LIN {X 0,Y 322.903,Z 1049.964,A -85,B 0,C 180,E1 13541.731,E2 13541.731} C_VEL
LIN {X 0,Y 332.533,Z 1032.411,A -85,B 0,C 180,E1 13538.987,E2 13538.987} C_VEL
LIN {X 0,Y 341.786,Z 1014.049,A -85,B 0,C 180,E1 13536.641,E2 13536.641} C_VEL
LIN {X 0,Y 350.913,Z 994.604,A -85,B 0,C 180,E1 13534.565,E2 13534.565} C_VEL
LIN {X 0,Y 358.946,Z 975.482,A -85,B 0,C 180,E1 13532.888,E2 13532.888} C_VEL
LIN {X 0,Y 366.893,Z 954.723,A -85,B 0,C 180,E1 13531.368,E2 13531.368} C_VEL
LIN {X 0,Y 373.86,Z 933.503,A -85,B 0,C 180,E1 13530.106,E2 13530.106} C_VEL
LIN {X 0,Y 380.358,Z 910.815,A -85,B 0,C 180,E1 13529.008,E2 13529.008} C_VEL
LIN {X 0,Y 385.815,Z 887.235,A -85,B 0,C 180,E1 13528.129,E2 13528.129} C_VEL
LIN {X 0,Y 390.273,Z 863.229,A -85,B 0,C 180,E1 13527.442,E2 13527.442} C_VEL
LIN {X 0,Y 393.285,Z 839.012,A -85,B 0,C 180,E1 13526.936,E2 13526.936} C_VEL
LIN {X 0,Y 410.602,Z 627.439,A -85,B 0,C 180,E1 13523.387,E2 13523.387} C_VEL
LIN {X 0,Y 404.165,Z 615.635,A -85,B 0,C 180,E1 13520.832,E2 13520.832} C_VEL
LIN {X 0,Y 397.85,Z 604.757,A -85,B 0,C 180,E1 13517.969,E2 13517.969} C_VEL
LIN {X 0,Y 392.489,Z 596.179,A -85,B 0,C 180,E1 13515.137,E2 13515.137} C_VEL
LIN {X 0,Y 387.858,Z 589.138,A -85,B 0,C 180,E1 13512.204,E2 13512.204} C_VEL
LIN {X 0,Y 384.835,Z 584.731,A -85,B 0,C 180,E1 13509.874,E2 13509.874} C_VEL
LIN {X 0,Y 381.69,Z 580.189,A -85,B 0,C 180,E1 13506.77,E2 13506.77} C_VEL
LIN {X 0,Y 378.64,Z 576.347,A -85,B 0,C 180,E1 13501.816,E2 13501.816} C_VEL
LIN {X 0,Y 377.972,Z 575.706,A -85,B 0,C 180,E1 13498.787,E2 13498.787} C_VEL
LIN {X 0,Y 378.254,Z 577.065,A -85,B 0,C 180,E1 13495.3,E2 13495.3} C_VEL
LIN {X 0,Y 380.09,Z 579.956,A -85,B 0,C 180,E1 13491.376,E2 13491.376} C_VEL
LIN {X 0,Y 382.905,Z 585.008,A -85,B 0,C 180,E1 13487.942,E2 13487.942} C_VEL
LIN {X 0,Y 385.173,Z 588.932,A -85,B 0,C 180,E1 13485.876,E2 13485.876} C_VEL
LIN {X 0,Y 388.941,Z 595.206,A -85,B 0,C 180,E1 13483.112,E2 13483.112} C_VEL
LIN {X 0,Y 394.171,Z 604.5,A -85,B 0,C 180,E1 13479.973,E2 13479.973} C_VEL
LIN {X 0,Y 400.396,Z 616.098,A -85,B 0,C 180,E1 13476.878,E2 13476.878} C_VEL
LIN {X 0,Y 406.234,Z 627.647,A -85,B 0,C 180,E1 13474.368,E2 13474.368} C_VEL
LIN {X 0,Y 409.258,Z 634.08,A -85,B 0,C 180,E1 13473.169,E2 13473.169} C_VEL
LIN {X 0,Y 392.663,Z 845.729,A -85,B 0,C 180,E1 13469.732,E2 13469.732} C_VEL
LIN {X 0,Y 389.223,Z 870.537,A -85,B 0,C 180,E1 13469.186,E2 13469.186} C_VEL
LIN {X 0,Y 384.954,Z 892.745,A -85,B 0,C 180,E1 13468.528,E2 13468.528} C_VEL
LIN {X 0,Y 379.397,Z 915.306,A -85,B 0,C 180,E1 13467.637,E2 13467.637} C_VEL
LIN {X 0,Y 373.122,Z 936.697,A -85,B 0,C 180,E1 13466.575,E2 13466.575} C_VEL
LIN {X 0,Y 365.655,Z 958.094,A -85,B 0,C 180,E1 13465.237,E2 13465.237} C_VEL
LIN {X 0,Y 357.495,Z 978.757,A -85,B 0,C 180,E1 13463.661,E2 13463.661} C_VEL
LIN {X 0,Y 348.897,Z 997.813,A -85,B 0,C 180,E1 13461.863,E2 13461.863} C_VEL
LIN {X 0,Y 339.99,Z 1016.009,A -85,B 0,C 180,E1 13459.8,E2 13459.8} C_VEL
LIN {X 0,Y 330.683,Z 1033.179,A -85,B 0,C 180,E1 13457.415,E2 13457.415} C_VEL
LIN {X 0,Y 321.318,Z 1049.45,A -85,B 0,C 180,E1 13454.691,E2 13454.691} C_VEL
LIN {X 0,Y 312.434,Z 1063.871,A -85,B 0,C 180,E1 13451.734,E2 13451.734} C_VEL
LIN {X 0,Y 303.544,Z 1077.822,A -85,B 0,C 180,E1 13448.264,E2 13448.264} C_VEL
LIN {X 0,Y 296.111,Z 1089.153,A -85,B 0,C 180,E1 13444.797,E2 13444.797} C_VEL
LIN {X 0,Y 288.785,Z 1100.377,A -85,B 0,C 180,E1 13440.596,E2 13440.596} C_VEL
LIN {X 0,Y 283.114,Z 1109.26,A -85,B 0,C 180,E1 13436.424,E2 13436.424} C_VEL
LIN {X 0,Y 278.099,Z 1117.701,A -85,B 0,C 180,E1 13431.373,E2 13431.373} C_VEL
LIN {X 0,Y 275.121,Z 1123.417,A -85,B 0,C 180,E1 13426.903,E2 13426.903} C_VEL
LIN {X 0,Y 273.116,Z 1128.104,A -85,B 0,C 180,E1 13421.831,E2 13421.831} C_VEL
LIN {X 0,Y 272.314,Z 1130.762,A -85,B 0,C 180,E1 13417.52,E2 13417.52} C_VEL
LIN {X 0,Y 272.028,Z 1132.355,A -85,B 0,C 180,E1 13412.739,E2 13412.739} C_VEL
LIN {X 0,Y 272.01,Z 1132.518,A -85,B 0,C 180,E1 13408.736,E2 13408.736} C_VEL
LIN {X 0,Y 272.117,Z 1131.71,A -85,B 0,C 180,E1 13404.729,E2 13404.729} C_VEL
LIN {X 0,Y 272.676,Z 1129.578,A -85,B 0,C 180,E1 13400.076,E2 13400.076} C_VEL
LIN {X 0,Y 274.088,Z 1125.684,A -85,B 0,C 180,E1 13395.205,E2 13395.205} C_VEL
LIN {X 0,Y 276.732,Z 1120.334,A -85,B 0,C 180,E1 13390.365,E2 13390.365} C_VEL
LIN {X 0,Y 280.577,Z 1113.483,A -85,B 0,C 180,E1 13385.806,E2 13385.806} C_VEL
LIN {X 0,Y 285.829,Z 1105.112,A -85,B 0,C 180,E1 13381.363,E2 13381.363} C_VEL
LIN {X 0,Y 292.154,Z 1095.285,A -85,B 0,C 180,E1 13377.265,E2 13377.265} C_VEL
LIN {X 0,Y 299.769,Z 1083.78,A -85,B 0,C 180,E1 13373.34,E2 13373.34} C_VEL
LIN {X 0,Y 307.712,Z 1071.486,A -85,B 0,C 180,E1 13369.955,E2 13369.955} C_VEL
LIN {X 0,Y 316.612,Z 1057.407,A -85,B 0,C 180,E1 13366.74,E2 13366.74} C_VEL
LIN {X 0,Y 325.483,Z 1042.519,A -85,B 0,C 180,E1 13363.97,E2 13363.97} C_VEL
LIN {X 0,Y 334.935,Z 1025.814,A -85,B 0,C 180,E1 13361.385,E2 13361.385} C_VEL
LIN {X 0,Y 343.865,Z 1008.56,A -85,B 0,C 180,E1 13359.201,E2 13359.201} C_VEL
LIN {X 0,Y 353.149,Z 989.023,A -85,B 0,C 180,E1 13357.153,E2 13357.153} C_VEL
LIN {X 0,Y 361.054,Z 970.43,A -85,B 0,C 180,E1 13355.561,E2 13355.561} C_VEL
LIN {X 0,Y 369.229,Z 948.778,A -85,B 0,C 180,E1 13354.038,E2 13354.038} C_VEL
LIN {X 0,Y 375.381,Z 929.911,A -85,B 0,C 180,E1 13352.959,E2 13352.959} C_VEL
LIN {X 0,Y 381.682,Z 907.48,A -85,B 0,C 180,E1 13351.92,E2 13351.92} C_VEL
LIN {X 0,Y 386.562,Z 885.839,A -85,B 0,C 180,E1 13351.142,E2 13351.142} C_VEL
LIN {X 0,Y 390.855,Z 861.566,A -85,B 0,C 180,E1 13350.489,E2 13350.489} C_VEL
LIN {X 0,Y 393.474,Z 839.331,A -85,B 0,C 180,E1 13350.048,E2 13350.048} C_VEL
LIN {X 0,Y 401.911,Z 730.436,A -85,B 0,C 180,E1 13348.274,E2 13348.274} C_VEL
LIN {X 0,Y 402.052,Z 722.869,A -85,B 0,C 180,E1 13348.025,E2 13348.025} C_VEL
LIN {X 0,Y 400.861,Z 703.163,A -85,B 0,C 180,E1 13346.9,E2 13346.9} C_VEL
LIN {X 0,Y 401.076,Z 696.654,A -85,B 0,C 180,E1 13346.702,E2 13346.702} C_VEL
LIN {X 0,Y 405.736,Z 638.185,A -85,B 0,C 180,E1 13345.744,E2 13345.744} C_VEL
LIN {X 0,Y 400.125,Z 626.654,A -85,B 0,C 180,E1 13343.334,E2 13343.334} C_VEL
LIN {X 0,Y 395.257,Z 617.143,A -85,B 0,C 180,E1 13340.975,E2 13340.975} C_VEL
LIN {X 0,Y 391.098,Z 609.419,A -85,B 0,C 180,E1 13338.676,E2 13338.676} C_VEL
LIN {X 0,Y 386.949,Z 601.81,A -85,B 0,C 180,E1 13335.974,E2 13335.974} C_VEL
LIN {X 0,Y 382.739,Z 594.401,A -85,B 0,C 180,E1 13332.523,E2 13332.523} C_VEL
LIN {X 0,Y 380.657,Z 590.854,A -85,B 0,C 180,E1 13330.289,E2 13330.289} C_VEL
LIN {X 0,Y 378.767,Z 587.132,A -85,B 0,C 180,E1 13327.432,E2 13327.432} C_VEL
LIN {X 0,Y 377.279,Z 584.215,A -85,B 0,C 180,E1 13321.974,E2 13321.974} C_VEL
LIN {X 0,Y 377.726,Z 584.352,A -85,B 0,C 180,E1 13318.938,E2 13318.938} C_VEL
LIN {X 0,Y 379.196,Z 586.5,A -85,B 0,C 180,E1 13315.614,E2 13315.614} C_VEL
LIN {X 0,Y 381.242,Z 588.925,A -85,B 0,C 180,E1 13312.919,E2 13312.919} C_VEL
LIN {X 0,Y 384.711,Z 594.101,A -85,B 0,C 180,E1 13309.593,E2 13309.593} C_VEL
LIN {X 0,Y 387.934,Z 599.004,A -85,B 0,C 180,E1 13307.193,E2 13307.193} C_VEL
LIN {X 0,Y 392.201,Z 605.658,A -85,B 0,C 180,E1 13304.549,E2 13304.549} C_VEL
LIN {X 0,Y 397.939,Z 615.402,A -85,B 0,C 180,E1 13301.543,E2 13301.543} C_VEL
LIN {X 0,Y 403.54,Z 625.439,A -85,B 0,C 180,E1 13299.02,E2 13299.02} C_VEL
LIN {X 0,Y 407.083,Z 632.137,A -85,B 0,C 180,E1 13297.567,E2 13297.567} C_VEL
LIN {X 0,Y 389.262,Z 843.506,A -85,B 0,C 180,E1 13294.032,E2 13294.032} C_VEL
LIN {X 0,Y 385.581,Z 869.279,A -85,B 0,C 180,E1 13293.455,E2 13293.455} C_VEL
LIN {X 0,Y 381.197,Z 891.496,A -85,B 0,C 180,E1 13292.795,E2 13292.795} C_VEL
LIN {X 0,Y 375.18,Z 915.552,A -85,B 0,C 180,E1 13291.854,E2 13291.854} C_VEL
LIN {X 0,Y 368.839,Z 936.823,A -85,B 0,C 180,E1 13290.8,E2 13290.8} C_VEL
LIN {X 0,Y 360.787,Z 959.799,A -85,B 0,C 180,E1 13289.376,E2 13289.376} C_VEL
LIN {X 0,Y 352.95,Z 979.483,A -85,B 0,C 180,E1 13287.893,E2 13287.893} C_VEL
LIN {X 0,Y 343.751,Z 1000.055,A -85,B 0,C 180,E1 13285.996,E2 13285.996} C_VEL
LIN {X 0,Y 334.941,Z 1018.035,A -85,B 0,C 180,E1 13284,E2 13284} C_VEL
LIN {X 0,Y 324.794,Z 1037.02,A -85,B 0,C 180,E1 13281.44,E2 13281.44} C_VEL
LIN {X 0,Y 315.852,Z 1052.706,A -85,B 0,C 180,E1 13278.889,E2 13278.889} C_VEL
LIN {X 0,Y 305.817,Z 1069.374,A -85,B 0,C 180,E1 13275.598,E2 13275.598} C_VEL
LIN {X 0,Y 297.663,Z 1082.472,A -85,B 0,C 180,E1 13272.469,E2 13272.469} C_VEL
LIN {X 0,Y 288.631,Z 1096.717,A -85,B 0,C 180,E1 13268.324,E2 13268.324} C_VEL
LIN {X 0,Y 281.666,Z 1107.82,A -85,B 0,C 180,E1 13264.363,E2 13264.363} C_VEL
LIN {X 0,Y 275.153,Z 1118.6,A -85,B 0,C 180,E1 13259.618,E2 13259.618} C_VEL
LIN {X 0,Y 270.803,Z 1126.415,A -85,B 0,C 180,E1 13255.36,E2 13255.36} C_VEL
LIN {X 0,Y 267.019,Z 1134.293,A -85,B 0,C 180,E1 13249.923,E2 13249.923} C_VEL
LIN {X 0,Y 265.197,Z 1139.135,A -85,B 0,C 180,E1 13245.527,E2 13245.527} C_VEL
LIN {X 0,Y 264.211,Z 1143.133,A -85,B 0,C 180,E1 13240.687,E2 13240.687} C_VEL
LIN {X 0,Y 263.966,Z 1145.544,A -85,B 0,C 180,E1 13235.87,E2 13235.87} C_VEL
LIN {X 0,Y 263.989,Z 1146.491,A -85,B 0,C 180,E1 13231.954,E2 13231.954} C_VEL
LIN {X 0,Y 263.992,Z 1146.511,A -85,B 0,C 180,E1 13228.264,E2 13228.264} C_VEL
LIN {X 0,Y 263.96,Z 1145.604,A -85,B 0,C 180,E1 13224.348,E2 13224.348} C_VEL
LIN {X 0,Y 264.164,Z 1143.39,A -85,B 0,C 180,E1 13219.752,E2 13219.752} C_VEL
LIN {X 0,Y 265.132,Z 1139.314,A -85,B 0,C 180,E1 13214.693,E2 13214.693} C_VEL
LIN {X 0,Y 267.017,Z 1134.249,A -85,B 0,C 180,E1 13210.076,E2 13210.076} C_VEL
LIN {X 0,Y 270.611,Z 1126.713,A -85,B 0,C 180,E1 13204.854,E2 13204.854} C_VEL
LIN {X 0,Y 275.146,Z 1118.526,A -85,B 0,C 180,E1 13200.381,E2 13200.381} C_VEL
LIN {X 0,Y 281.976,Z 1107.201,A -85,B 0,C 180,E1 13195.433,E2 13195.433} C_VEL
LIN {X 0,Y 289.002,Z 1096.026,A -85,B 0,C 180,E1 13191.481,E2 13191.481} C_VEL
LIN {X 0,Y 297.648,Z 1082.336,A -85,B 0,C 180,E1 13187.528,E2 13187.528} C_VEL
LIN {X 0,Y 306.039,Z 1068.835,A -85,B 0,C 180,E1 13184.314,E2 13184.314} C_VEL
LIN {X 0,Y 316.373,Z 1051.575,A -85,B 0,C 180,E1 13180.943,E2 13180.943} C_VEL
LIN {X 0,Y 325.579,Z 1035.387,A -85,B 0,C 180,E1 13178.343,E2 13178.343} C_VEL
LIN {X 0,Y 335.535,Z 1016.541,A -85,B 0,C 180,E1 13175.849,E2 13175.849} C_VEL
LIN {X 0,Y 344.173,Z 998.833,A -85,B 0,C 180,E1 13173.904,E2 13173.904} C_VEL
LIN {X 0,Y 353.597,Z 977.481,A -85,B 0,C 180,E1 13171.969,E2 13171.969} C_VEL
LIN {X 0,Y 361.109,Z 958.494,A -85,B 0,C 180,E1 13170.554,E2 13170.554} C_VEL
LIN {X 0,Y 369.167,Z 935.183,A -85,B 0,C 180,E1 13169.132,E2 13169.132} C_VEL
LIN {X 0,Y 375.263,Z 914.581,A -85,B 0,C 180,E1 13168.121,E2 13168.121} C_VEL
LIN {X 0,Y 381.465,Z 889.296,A -85,B 0,C 180,E1 13167.15,E2 13167.15} C_VEL
LIN {X 0,Y 385.776,Z 867.055,A -85,B 0,C 180,E1 13166.502,E2 13166.502} C_VEL
LIN {X 0,Y 389.241,Z 841.731,A -85,B 0,C 180,E1 13165.95,E2 13165.95} C_VEL
LIN {X 0,Y 406.871,Z 631.81,A -85,B 0,C 180,E1 13162.432,E2 13162.432} C_VEL
LIN {X 0,Y 399.929,Z 619.065,A -85,B 0,C 180,E1 13159.498,E2 13159.498} C_VEL
LIN {X 0,Y 393.816,Z 608.454,A -85,B 0,C 180,E1 13156.483,E2 13156.483} C_VEL
LIN {X 0,Y 388.661,Z 600.303,A -85,B 0,C 180,E1 13153.464,E2 13153.464} C_VEL
LIN {X 0,Y 386.042,Z 596.274,A -85,B 0,C 180,E1 13151.656,E2 13151.656} C_VEL
LIN {X 0,Y 383.497,Z 592.425,A -85,B 0,C 180,E1 13149.606,E2 13149.606} C_VEL
LIN {X 0,Y 380.576,Z 588.062,A -85,B 0,C 180,E1 13146.638,E2 13146.638} C_VEL
LIN {X 0,Y 377.61,Z 584.234,A -85,B 0,C 180,E1 13141.669,E2 13141.669} C_VEL
LIN {X 0,Y 376.986,Z 583.655,A -85,B 0,C 180,E1 13138.632,E2 13138.632} C_VEL
LIN {X 0,Y 377.318,Z 585.14,A -85,B 0,C 180,E1 13135.135,E2 13135.135} C_VEL
LIN {X 0,Y 378.967,Z 587.768,A -85,B 0,C 180,E1 13131.58,E2 13131.58} C_VEL
LIN {X 0,Y 381.708,Z 592.841,A -85,B 0,C 180,E1 13128.133,E2 13128.133} C_VEL
LIN {X 0,Y 383.842,Z 596.653,A -85,B 0,C 180,E1 13126.134,E2 13126.134} C_VEL
LIN {X 0,Y 387.417,Z 602.767,A -85,B 0,C 180,E1 13123.43,E2 13123.43} C_VEL
LIN {X 0,Y 392.719,Z 612.462,A -85,B 0,C 180,E1 13120.168,E2 13120.168} C_VEL
LIN {X 0,Y 398.552,Z 623.768,A -85,B 0,C 180,E1 13117.194,E2 13117.194} C_VEL
LIN {X 0,Y 403.876,Z 634.566,A -85,B 0,C 180,E1 13114.836,E2 13114.836} C_VEL
LIN {X 0,Y 405.574,Z 638.42,A -85,B 0,C 180,E1 13114.126,E2 13114.126} C_VEL
LIN {X 0,Y 388.882,Z 845.735,A -85,B 0,C 180,E1 13110.768,E2 13110.768} C_VEL
LIN {X 0,Y 385.368,Z 870.544,A -85,B 0,C 180,E1 13110.226,E2 13110.226} C_VEL
LIN {X 0,Y 381.009,Z 892.763,A -85,B 0,C 180,E1 13109.574,E2 13109.574} C_VEL
LIN {X 0,Y 375.184,Z 915.866,A -85,B 0,C 180,E1 13108.667,E2 13108.667} C_VEL
LIN {X 0,Y 368.789,Z 937.151,A -85,B 0,C 180,E1 13107.614,E2 13107.614} C_VEL
LIN {X 0,Y 361.097,Z 958.617,A -85,B 0,C 180,E1 13106.274,E2 13106.274} C_VEL
LIN {X 0,Y 352.79,Z 979.102,A -85,B 0,C 180,E1 13104.713,E2 13104.713} C_VEL
LIN {X 0,Y 344.01,Z 998.066,A -85,B 0,C 180,E1 13102.926,E2 13102.926} C_VEL
LIN {X 0,Y 334.655,Z 1016.609,A -85,B 0,C 180,E1 13100.816,E2 13100.816} C_VEL
LIN {X 0,Y 325.255,Z 1033.454,A -85,B 0,C 180,E1 13098.466,E2 13098.466} C_VEL
LIN {X 0,Y 315.594,Z 1049.705,A -85,B 0,C 180,E1 13095.728,E2 13095.728} C_VEL
LIN {X 0,Y 306.483,Z 1064.007,A -85,B 0,C 180,E1 13092.772,E2 13092.772} C_VEL
LIN {X 0,Y 297.185,Z 1078.057,A -85,B 0,C 180,E1 13089.237,E2 13089.237} C_VEL
LIN {X 0,Y 289.444,Z 1089.384,A -85,B 0,C 180,E1 13085.719,E2 13085.719} C_VEL
LIN {X 0,Y 281.786,Z 1100.601,A -85,B 0,C 180,E1 13081.441,E2 13081.441} C_VEL
LIN {X 0,Y 275.83,Z 1109.483,A -85,B 0,C 180,E1 13077.178,E2 13077.178} C_VEL
LIN {X 0,Y 270.645,Z 1117.731,A -85,B 0,C 180,E1 13072.138,E2 13072.138} C_VEL
LIN {X 0,Y 267.456,Z 1123.446,A -85,B 0,C 180,E1 13067.574,E2 13067.574} C_VEL
LIN {X 0,Y 265.208,Z 1128.316,A -85,B 0,C 180,E1 13062.189,E2 13062.189} C_VEL
LIN {X 0,Y 264.353,Z 1130.934,A -85,B 0,C 180,E1 13057.826,E2 13057.826} C_VEL
LIN {X 0,Y 264.038,Z 1132.544,A -85,B 0,C 180,E1 13053.039,E2 13053.039} C_VEL
LIN {X 0,Y 264.013,Z 1132.728,A -85,B 0,C 180,E1 13048.698,E2 13048.698} C_VEL
LIN {X 0,Y 264.13,Z 1131.92,A -85,B 0,C 180,E1 13044.569,E2 13044.569} C_VEL
LIN {X 0,Y 264.728,Z 1129.79,A -85,B 0,C 180,E1 13039.775,E2 13039.775} C_VEL
LIN {X 0,Y 266.256,Z 1125.898,A -85,B 0,C 180,E1 13034.759,E2 13034.759} C_VEL
LIN {X 0,Y 269.081,Z 1120.55,A -85,B 0,C 180,E1 13029.783,E2 13029.783} C_VEL
LIN {X 0,Y 273.156,Z 1113.7,A -85,B 0,C 180,E1 13025.105,E2 13025.105} C_VEL
LIN {X 0,Y 278.688,Z 1105.334,A -85,B 0,C 180,E1 13020.558,E2 13020.558} C_VEL
LIN {X 0,Y 285.316,Z 1095.51,A -85,B 0,C 180,E1 13016.378,E2 13016.378} C_VEL
LIN {X 0,Y 293.265,Z 1084.013,A -85,B 0,C 180,E1 13012.388,E2 13012.388} C_VEL
LIN {X 0,Y 301.516,Z 1071.722,A -85,B 0,C 180,E1 13008.958,E2 13008.958} C_VEL
LIN {X 0,Y 310.74,Z 1057.658,A -85,B 0,C 180,E1 13005.712,E2 13005.712} C_VEL
LIN {X 0,Y 319.752,Z 1043.028,A -85,B 0,C 180,E1 13002.967,E2 13002.967} C_VEL
LIN {X 0,Y 329.453,Z 1026.447,A -85,B 0,C 180,E1 13000.378,E2 13000.378} C_VEL
LIN {X 0,Y 338.819,Z 1008.855,A -85,B 0,C 180,E1 12998.143,E2 12998.143} C_VEL
LIN {X 0,Y 348.023,Z 990.085,A -85,B 0,C 180,E1 12996.164,E2 12996.164} C_VEL
LIN {X 0,Y 356.36,Z 970.988,A -85,B 0,C 180,E1 12994.526,E2 12994.526} C_VEL
LIN {X 0,Y 364.462,Z 950.207,A -85,B 0,C 180,E1 12993.056,E2 12993.056} C_VEL
LIN {X 0,Y 371.092,Z 930.392,A -85,B 0,C 180,E1 12991.923,E2 12991.923} C_VEL
LIN {X 0,Y 377.525,Z 908.106,A -85,B 0,C 180,E1 12990.893,E2 12990.893} C_VEL
LIN {X 0,Y 382.609,Z 886.081,A -85,B 0,C 180,E1 12990.105,E2 12990.105} C_VEL
LIN {X 0,Y 386.974,Z 862.046,A -85,B 0,C 180,E1 12989.461,E2 12989.461} C_VEL
LIN {X 0,Y 389.69,Z 839.602,A -85,B 0,C 180,E1 12989.017,E2 12989.017} C_VEL
LIN {X 0,Y 401.076,Z 696.654,A -85,B 0,C 180,E1 12986.702,E2 12986.702} C_VEL
LIN {X 0,Y 401.28,Z 689.088,A -85,B 0,C 180,E1 12986.456,E2 12986.456} C_VEL
LIN {X 0,Y 400.308,Z 669.401,A -85,B 0,C 180,E1 12985.318,E2 12985.318} C_VEL
LIN {X 0,Y 400.547,Z 662.896,A -85,B 0,C 180,E1 12985.115,E2 12985.115} C_VEL
LIN {X 0,Y 402.173,Z 642.482,A -85,B 0,C 180,E1 12984.767,E2 12984.767} C_VEL
LIN {X 0,Y 396.956,Z 631.632,A -85,B 0,C 180,E1 12982.395,E2 12982.395} C_VEL
LIN {X 0,Y 392.14,Z 622.064,A -85,B 0,C 180,E1 12979.902,E2 12979.902} C_VEL
LIN {X 0,Y 387.97,Z 614.013,A -85,B 0,C 180,E1 12977.395,E2 12977.395} C_VEL
LIN {X 0,Y 384.024,Z 606.829,A -85,B 0,C 180,E1 12974.552,E2 12974.552} C_VEL
LIN {X 0,Y 381.229,Z 601.727,A -85,B 0,C 180,E1 12972.035,E2 12972.035} C_VEL
LIN {X 0,Y 379.441,Z 598.565,A -85,B 0,C 180,E1 12970.016,E2 12970.016} C_VEL
LIN {X 0,Y 377.634,Z 594.913,A -85,B 0,C 180,E1 12967.149,E2 12967.149} C_VEL
LIN {X 0,Y 376.306,Z 592.121,A -85,B 0,C 180,E1 12961.827,E2 12961.827} C_VEL
LIN {X 0,Y 376.75,Z 592.304,A -85,B 0,C 180,E1 12958.936,E2 12958.936} C_VEL
LIN {X 0,Y 378.309,Z 594.631,A -85,B 0,C 180,E1 12955.452,E2 12955.452} C_VEL
LIN {X 0,Y 380.058,Z 596.726,A -85,B 0,C 180,E1 12953.125,E2 12953.125} C_VEL
LIN {X 0,Y 383.355,Z 601.786,A -85,B 0,C 180,E1 12949.86,E2 12949.86} C_VEL
LIN {X 0,Y 386.504,Z 606.712,A -85,B 0,C 180,E1 12947.449,E2 12947.449} C_VEL
LIN {X 0,Y 390.619,Z 613.327,A -85,B 0,C 180,E1 12944.827,E2 12944.827} C_VEL
LIN {X 0,Y 396.255,Z 623.12,A -85,B 0,C 180,E1 12941.804,E2 12941.804} C_VEL
LIN {X 0,Y 402.628,Z 634.926,A -85,B 0,C 180,E1 12938.894,E2 12938.894} C_VEL
LIN {X 0,Y 403.466,Z 636.791,A -85,B 0,C 180,E1 12938.529,E2 12938.529} C_VEL
LIN {X 0,Y 385.611,Z 843.606,A -85,B 0,C 180,E1 12935.087,E2 12935.087} C_VEL
LIN {X 0,Y 381.867,Z 869.298,A -85,B 0,C 180,E1 12934.516,E2 12934.516} C_VEL
LIN {X 0,Y 377.399,Z 891.516,A -85,B 0,C 180,E1 12933.863,E2 12933.863} C_VEL
LIN {X 0,Y 371.534,Z 914.61,A -85,B 0,C 180,E1 12932.975,E2 12932.975} C_VEL
LIN {X 0,Y 365.305,Z 935.197,A -85,B 0,C 180,E1 12931.974,E2 12931.974} C_VEL
LIN {X 0,Y 357.061,Z 958.492,A -85,B 0,C 180,E1 12930.564,E2 12930.564} C_VEL
LIN {X 0,Y 349.366,Z 977.477,A -85,B 0,C 180,E1 12929.161,E2 12929.161} C_VEL
LIN {X 0,Y 339.903,Z 998.385,A -85,B 0,C 180,E1 12927.281,E2 12927.281} C_VEL
LIN {X 0,Y 331.133,Z 1015.886,A -85,B 0,C 180,E1 12925.371,E2 12925.371} C_VEL
LIN {X 0,Y 320.926,Z 1034.688,A -85,B 0,C 180,E1 12922.902,E2 12922.902} C_VEL
LIN {X 0,Y 311.607,Z 1050.559,A -85,B 0,C 180,E1 12920.365,E2 12920.365} C_VEL
LIN {X 0,Y 301.359,Z 1067.174,A -85,B 0,C 180,E1 12917.161,E2 12917.161} C_VEL
LIN {X 0,Y 292.515,Z 1080.801,A -85,B 0,C 180,E1 12913.94,E2 12913.94} C_VEL
LIN {X 0,Y 283.699,Z 1094.262,A -85,B 0,C 180,E1 12910.109,E2 12910.109} C_VEL
LIN {X 0,Y 275.869,Z 1106.008,A -85,B 0,C 180,E1 12905.957,E2 12905.957} C_VEL
LIN {X 0,Y 269.062,Z 1116.71,A -85,B 0,C 180,E1 12901.35,E2 12901.35} C_VEL
LIN {X 0,Y 263.71,Z 1125.562,A -85,B 0,C 180,E1 12896.514,E2 12896.514} C_VEL
LIN {X 0,Y 259.761,Z 1133.159,A -85,B 0,C 180,E1 12891.326,E2 12891.326} C_VEL
LIN {X 0,Y 257.401,Z 1138.704,A -85,B 0,C 180,E1 12886.242,E2 12886.242} C_VEL
LIN {X 0,Y 256.306,Z 1142.587,A -85,B 0,C 180,E1 12881.476,E2 12881.476} C_VEL
LIN {X 0,Y 255.977,Z 1145.262,A -85,B 0,C 180,E1 12876.279,E2 12876.279} C_VEL
LIN {X 0,Y 255.984,Z 1146.257,A -85,B 0,C 180,E1 12872.239,E2 12872.239} C_VEL
LIN {X 0,Y 255.997,Z 1146.325,A -85,B 0,C 180,E1 12868.433,E2 12868.433} C_VEL
LIN {X 0,Y 255.957,Z 1145.536,A -85,B 0,C 180,E1 12864.62,E2 12864.62} C_VEL
LIN {X 0,Y 256.091,Z 1143.774,A -85,B 0,C 180,E1 12860.562,E2 12860.562} C_VEL
LIN {X 0,Y 256.938,Z 1140.171,A -85,B 0,C 180,E1 12855.348,E2 12855.348} C_VEL
LIN {X 0,Y 258.825,Z 1135.085,A -85,B 0,C 180,E1 12850.361,E2 12850.361} C_VEL
LIN {X 0,Y 262.21,Z 1128.284,A -85,B 0,C 180,E1 12845.199,E2 12845.199} C_VEL
LIN {X 0,Y 267.198,Z 1119.55,A -85,B 0,C 180,E1 12840.152,E2 12840.152} C_VEL
LIN {X 0,Y 273.539,Z 1109.596,A -85,B 0,C 180,E1 12835.487,E2 12835.487} C_VEL
LIN {X 0,Y 281.053,Z 1098.019,A -85,B 0,C 180,E1 12831.181,E2 12831.181} C_VEL
LIN {X 0,Y 289.778,Z 1084.947,A -85,B 0,C 180,E1 12827.175,E2 12827.175} C_VEL
LIN {X 0,Y 298.793,Z 1070.937,A -85,B 0,C 180,E1 12823.711,E2 12823.711} C_VEL
LIN {X 0,Y 308.804,Z 1055.068,A -85,B 0,C 180,E1 12820.455,E2 12820.455} C_VEL
LIN {X 0,Y 318.807,Z 1038.071,A -85,B 0,C 180,E1 12817.633,E2 12817.633} C_VEL
LIN {X 0,Y 328.897,Z 1019.931,A -85,B 0,C 180,E1 12815.135,E2 12815.135} C_VEL
LIN {X 0,Y 338.29,Z 1001.314,A -85,B 0,C 180,E1 12813.042,E2 12813.042} C_VEL
LIN {X 0,Y 347.588,Z 981.284,A -85,B 0,C 180,E1 12811.167,E2 12811.167} C_VEL
LIN {X 0,Y 356.067,Z 960.558,A -85,B 0,C 180,E1 12809.598,E2 12809.598} C_VEL
LIN {X 0,Y 363.831,Z 939.237,A -85,B 0,C 180,E1 12808.26,E2 12808.26} C_VEL
LIN {X 0,Y 370.767,Z 916.599,A -85,B 0,C 180,E1 12807.133,E2 12807.133} C_VEL
LIN {X 0,Y 376.882,Z 892.996,A -85,B 0,C 180,E1 12806.203,E2 12806.203} C_VEL
LIN {X 0,Y 381.508,Z 870.155,A -85,B 0,C 180,E1 12805.523,E2 12805.523} C_VEL
LIN {X 0,Y 385.215,Z 845.424,A -85,B 0,C 180,E1 12804.963,E2 12804.963} C_VEL
LIN {X 0,Y 392.431,Z 762.771,A -85,B 0,C 180,E1 12803.556,E2 12803.556} C_VEL
LIN {X 0,Y 403.238,Z 636.332,A -85,B 0,C 180,E1 12801.461,E2 12801.461} C_VEL
LIN {X 0,Y 396.888,Z 624.491,A -85,B 0,C 180,E1 12798.622,E2 12798.622} C_VEL
LIN {X 0,Y 391.558,Z 615.089,A -85,B 0,C 180,E1 12795.857,E2 12795.857} C_VEL
LIN {X 0,Y 386.99,Z 607.667,A -85,B 0,C 180,E1 12793.066,E2 12793.066} C_VEL
LIN {X 0,Y 384.456,Z 603.677,A -85,B 0,C 180,E1 12791.248,E2 12791.248} C_VEL
LIN {X 0,Y 382.082,Z 600.017,A -85,B 0,C 180,E1 12789.262,E2 12789.262} C_VEL
LIN {X 0,Y 379.337,Z 595.811,A -85,B 0,C 180,E1 12786.356,E2 12786.356} C_VEL
LIN {X 0,Y 376.582,Z 592.121,A -85,B 0,C 180,E1 12781.521,E2 12781.521} C_VEL
LIN {X 0,Y 376.012,Z 591.596,A -85,B 0,C 180,E1 12778.629,E2 12778.629} C_VEL
LIN {X 0,Y 376.357,Z 593.164,A -85,B 0,C 180,E1 12775.064,E2 12775.064} C_VEL
LIN {X 0,Y 377.869,Z 595.629,A -85,B 0,C 180,E1 12771.753,E2 12771.753} C_VEL
LIN {X 0,Y 380.443,Z 600.538,A -85,B 0,C 180,E1 12768.401,E2 12768.401} C_VEL
LIN {X 0,Y 382.436,Z 604.207,A -85,B 0,C 180,E1 12766.467,E2 12766.467} C_VEL
LIN {X 0,Y 385.85,Z 610.249,A -85,B 0,C 180,E1 12763.786,E2 12763.786} C_VEL
LIN {X 0,Y 390.895,Z 619.732,A -85,B 0,C 180,E1 12760.577,E2 12760.577} C_VEL
LIN {X 0,Y 396.578,Z 631.12,A -85,B 0,C 180,E1 12757.583,E2 12757.583} C_VEL
LIN {X 0,Y 401.705,Z 641.813,A -85,B 0,C 180,E1 12755.241,E2 12755.241} C_VEL
LIN {X 0,Y 402,Z 642.783,A -85,B 0,C 180,E1 12755.1,E2 12755.1} C_VEL
LIN {X 0,Y 385.229,Z 845.77,A -85,B 0,C 180,E1 12751.824,E2 12751.824} C_VEL
LIN {X 0,Y 381.641,Z 870.552,A -85,B 0,C 180,E1 12751.287,E2 12751.287} C_VEL
LIN {X 0,Y 377.174,Z 892.874,A -85,B 0,C 180,E1 12750.639,E2 12750.639} C_VEL
LIN {X 0,Y 371.46,Z 915.149,A -85,B 0,C 180,E1 12749.776,E2 12749.776} C_VEL
LIN {X 0,Y 364.953,Z 936.432,A -85,B 0,C 180,E1 12748.739,E2 12748.739} C_VEL
LIN {X 0,Y 357.159,Z 957.868,A -85,B 0,C 180,E1 12747.424,E2 12747.424} C_VEL
LIN {X 0,Y 348.888,Z 977.921,A -85,B 0,C 180,E1 12745.92,E2 12745.92} C_VEL
LIN {X 0,Y 340.064,Z 996.667,A -85,B 0,C 180,E1 12744.188,E2 12744.188} C_VEL
LIN {X 0,Y 330.907,Z 1014.511,A -85,B 0,C 180,E1 12742.201,E2 12742.201} C_VEL
LIN {X 0,Y 320.827,Z 1032.227,A -85,B 0,C 180,E1 12739.78,E2 12739.78} C_VEL
LIN {X 0,Y 311.079,Z 1048.263,A -85,B 0,C 180,E1 12737.126,E2 12737.126} C_VEL
LIN {X 0,Y 301.497,Z 1062.852,A -85,B 0,C 180,E1 12734.143,E2 12734.143} C_VEL
LIN {X 0,Y 292.295,Z 1076.394,A -85,B 0,C 180,E1 12730.797,E2 12730.797} C_VEL
LIN {X 0,Y 283.653,Z 1088.493,A -85,B 0,C 180,E1 12727.07,E2 12727.07} C_VEL
LIN {X 0,Y 275.865,Z 1099.474,A -85,B 0,C 180,E1 12722.935,E2 12722.935} C_VEL
LIN {X 0,Y 269.132,Z 1108.914,A -85,B 0,C 180,E1 12718.395,E2 12718.395} C_VEL
LIN {X 0,Y 263.702,Z 1117.066,A -85,B 0,C 180,E1 12713.462,E2 12713.462} C_VEL
LIN {X 0,Y 260.013,Z 1123.112,A -85,B 0,C 180,E1 12708.613,E2 12708.613} C_VEL
LIN {X 0,Y 257.529,Z 1128.069,A -85,B 0,C 180,E1 12703.243,E2 12703.243} C_VEL
LIN {X 0,Y 256.451,Z 1130.927,A -85,B 0,C 180,E1 12698.52,E2 12698.52} C_VEL
LIN {X 0,Y 256.062,Z 1132.613,A -85,B 0,C 180,E1 12693.806,E2 12693.806} C_VEL
LIN {X 0,Y 256.016,Z 1132.967,A -85,B 0,C 180,E1 12688.956,E2 12688.956} C_VEL
LIN {X 0,Y 256.13,Z 1132.195,A -85,B 0,C 180,E1 12684.624,E2 12684.624} C_VEL
LIN {X 0,Y 256.708,Z 1130.231,A -85,B 0,C 180,E1 12679.905,E2 12679.905} C_VEL
LIN {X 0,Y 258.247,Z 1126.509,A -85,B 0,C 180,E1 12674.735,E2 12674.735} C_VEL
LIN {X 0,Y 260.976,Z 1121.532,A -85,B 0,C 180,E1 12669.829,E2 12669.829} C_VEL
LIN {X 0,Y 265.409,Z 1114.471,A -85,B 0,C 180,E1 12664.712,E2 12664.712} C_VEL
LIN {X 0,Y 271.047,Z 1106.33,A -85,B 0,C 180,E1 12660.102,E2 12660.102} C_VEL
LIN {X 0,Y 278.19,Z 1096.238,A -85,B 0,C 180,E1 12655.646,E2 12655.646} C_VEL
LIN {X 0,Y 286.423,Z 1084.862,A -85,B 0,C 180,E1 12651.582,E2 12651.582} C_VEL
LIN {X 0,Y 295.415,Z 1071.958,A -85,B 0,C 180,E1 12647.92,E2 12647.92} C_VEL
LIN {X 0,Y 304.971,Z 1057.908,A -85,B 0,C 180,E1 12644.645,E2 12644.645} C_VEL
LIN {X 0,Y 314.277,Z 1043.286,A -85,B 0,C 180,E1 12641.885,E2 12641.885} C_VEL
LIN {X 0,Y 324.269,Z 1026.727,A -85,B 0,C 180,E1 12639.288,E2 12639.288} C_VEL
LIN {X 0,Y 333.892,Z 1009.149,A -85,B 0,C 180,E1 12637.053,E2 12637.053} C_VEL
LIN {X 0,Y 343.333,Z 990.419,A -85,B 0,C 180,E1 12635.079,E2 12635.079} C_VEL
LIN {X 0,Y 351.783,Z 971.549,A -85,B 0,C 180,E1 12633.464,E2 12633.464} C_VEL
LIN {X 0,Y 360.155,Z 950.638,A -85,B 0,C 180,E1 12631.988,E2 12631.988} C_VEL
LIN {X 0,Y 366.927,Z 930.872,A -85,B 0,C 180,E1 12630.863,E2 12630.863} C_VEL
LIN {X 0,Y 373.493,Z 908.731,A -85,B 0,C 180,E1 12629.843,E2 12629.843} C_VEL
LIN {X 0,Y 378.746,Z 886.49,A -85,B 0,C 180,E1 12629.053,E2 12629.053} C_VEL
LIN {X 0,Y 383.173,Z 862.843,A -85,B 0,C 180,E1 12628.419,E2 12628.419} C_VEL
LIN {X 0,Y 386.018,Z 840.02,A -85,B 0,C 180,E1 12627.968,E2 12627.968} C_VEL
LIN {X 0,Y 400.547,Z 662.896,A -85,B 0,C 180,E1 12625.115,E2 12625.115} C_VEL
LIN {X 0,Y 400.592,Z 657.662,A -85,B 0,C 180,E1 12624.902,E2 12624.902} C_VEL
LIN {X 0,Y 399.843,Z 652.089,A -85,B 0,C 180,E1 12624.401,E2 12624.401} C_VEL
LIN {X 0,Y 398.281,Z 646.623,A -85,B 0,C 180,E1 12623.604,E2 12623.604} C_VEL
LIN {X 0,Y 394.621,Z 638.162,A -85,B 0,C 180,E1 12621.812,E2 12621.812} C_VEL
LIN {X 0,Y 394.342,Z 637.548,A -85,B 0,C 180,E1 12621.67,E2 12621.67} C_VEL
LIN {X 0,Y 388.987,Z 626.542,A -85,B 0,C 180,E1 12618.704,E2 12618.704} C_VEL
LIN {X 0,Y 384.273,Z 617.457,A -85,B 0,C 180,E1 12615.546,E2 12615.546} C_VEL
LIN {X 0,Y 380.327,Z 610.038,A -85,B 0,C 180,E1 12612.141,E2 12612.141} C_VEL
LIN {X 0,Y 378.233,Z 606.276,A -85,B 0,C 180,E1 12609.741,E2 12609.741} C_VEL
LIN {X 0,Y 376.588,Z 602.797,A -85,B 0,C 180,E1 12607.015,E2 12607.015} C_VEL
LIN {X 0,Y 375.335,Z 600.029,A -85,B 0,C 180,E1 12601.679,E2 12601.679} C_VEL
LIN {X 0,Y 375.817,Z 600.321,A -85,B 0,C 180,E1 12598.78,E2 12598.78} C_VEL
LIN {X 0,Y 378.707,Z 604.166,A -85,B 0,C 180,E1 12593.557,E2 12593.557} C_VEL
LIN {X 0,Y 382.008,Z 609.471,A -85,B 0,C 180,E1 12590.128,E2 12590.128} C_VEL
LIN {X 0,Y 385.082,Z 614.419,A -85,B 0,C 180,E1 12587.707,E2 12587.707} C_VEL
LIN {X 0,Y 389.047,Z 620.991,A -85,B 0,C 180,E1 12585.107,E2 12585.107} C_VEL
LIN {X 0,Y 394.441,Z 630.602,A -85,B 0,C 180,E1 12582.138,E2 12582.138} C_VEL
LIN {X 0,Y 399.977,Z 641.285,A -85,B 0,C 180,E1 12579.511,E2 12579.511} C_VEL
LIN {X 0,Y 382.094,Z 843.715,A -85,B 0,C 180,E1 12576.161,E2 12576.161} C_VEL
LIN {X 0,Y 378.263,Z 869.448,A -85,B 0,C 180,E1 12575.595,E2 12575.595} C_VEL
LIN {X 0,Y 373.711,Z 891.649,A -85,B 0,C 180,E1 12574.95,E2 12574.95} C_VEL
LIN {X 0,Y 367.54,Z 915.356,A -85,B 0,C 180,E1 12574.043,E2 12574.043} C_VEL
LIN {X 0,Y 360.779,Z 937.102,A -85,B 0,C 180,E1 12572.986,E2 12572.986} C_VEL
LIN {X 0,Y 352.738,Z 959.067,A -85,B 0,C 180,E1 12571.65,E2 12571.65} C_VEL
LIN {X 0,Y 344.933,Z 977.847,A -85,B 0,C 180,E1 12570.266,E2 12570.266} C_VEL
LIN {X 0,Y 334.863,Z 999.418,A -85,B 0,C 180,E1 12568.321,E2 12568.321} C_VEL
LIN {X 0,Y 325.882,Z 1016.816,A -85,B 0,C 180,E1 12566.412,E2 12566.412} C_VEL
LIN {X 0,Y 314.783,Z 1036.478,A -85,B 0,C 180,E1 12563.785,E2 12563.785} C_VEL
LIN {X 0,Y 305.245,Z 1052.177,A -85,B 0,C 180,E1 12561.226,E2 12561.226} C_VEL
LIN {X 0,Y 294.193,Z 1069.279,A -85,B 0,C 180,E1 12557.811,E2 12557.811} C_VEL
LIN {X 0,Y 285.162,Z 1082.701,A -85,B 0,C 180,E1 12554.53,E2 12554.53} C_VEL
LIN {X 0,Y 275.604,Z 1096.529,A -85,B 0,C 180,E1 12550.37,E2 12550.37} C_VEL
LIN {X 0,Y 268.034,Z 1107.494,A -85,B 0,C 180,E1 12546.314,E2 12546.314} C_VEL
LIN {X 0,Y 260.873,Z 1118.154,A -85,B 0,C 180,E1 12541.418,E2 12541.418} C_VEL
LIN {X 0,Y 255.961,Z 1125.972,A -85,B 0,C 180,E1 12536.946,E2 12536.946} C_VEL
LIN {X 0,Y 251.618,Z 1133.859,A -85,B 0,C 180,E1 12531.2,E2 12531.2} C_VEL
LIN {X 0,Y 249.476,Z 1138.704,A -85,B 0,C 180,E1 12526.533,E2 12526.533} C_VEL
LIN {X 0,Y 248.289,Z 1142.706,A -85,B 0,C 180,E1 12521.381,E2 12521.381} C_VEL
LIN {X 0,Y 247.978,Z 1145.123,A -85,B 0,C 180,E1 12516.25,E2 12516.25} C_VEL
LIN {X 0,Y 247.991,Z 1146.071,A -85,B 0,C 180,E1 12512.08,E2 12512.08} C_VEL
LIN {X 0,Y 247.999,Z 1146.115,A -85,B 0,C 180,E1 12508.383,E2 12508.383} C_VEL
LIN {X 0,Y 247.961,Z 1145.325,A -85,B 0,C 180,E1 12504.446,E2 12504.446} C_VEL
LIN {X 0,Y 248.134,Z 1143.441,A -85,B 0,C 180,E1 12500.022,E2 12500.022} C_VEL
LIN {X 0,Y 249.196,Z 1139.489,A -85,B 0,C 180,E1 12494.365,E2 12494.365} C_VEL
LIN {X 0,Y 251.223,Z 1134.602,A -85,B 0,C 180,E1 12489.497,E2 12489.497} C_VEL
LIN {X 0,Y 254.933,Z 1127.723,A -85,B 0,C 180,E1 12484.192,E2 12484.192} C_VEL
LIN {X 0,Y 260.043,Z 1119.325,A -85,B 0,C 180,E1 12479.243,E2 12479.243} C_VEL
LIN {X 0,Y 266.868,Z 1109.17,A -85,B 0,C 180,E1 12474.395,E2 12474.395} C_VEL
LIN {X 0,Y 274.553,Z 1097.899,A -85,B 0,C 180,E1 12470.135,E2 12470.135} C_VEL
LIN {X 0,Y 283.742,Z 1084.7,A -85,B 0,C 180,E1 12466.035,E2 12466.035} C_VEL
LIN {X 0,Y 293.467,Z 1070.175,A -85,B 0,C 180,E1 12462.425,E2 12462.425} C_VEL
LIN {X 0,Y 303.713,Z 1054.454,A -85,B 0,C 180,E1 12459.206,E2 12459.206} C_VEL
LIN {X 0,Y 313.878,Z 1037.729,A -85,B 0,C 180,E1 12456.432,E2 12456.432} C_VEL
LIN {X 0,Y 324.393,Z 1019.322,A -85,B 0,C 180,E1 12453.911,E2 12453.911} C_VEL
LIN {X 0,Y 333.821,Z 1001.132,A -85,B 0,C 180,E1 12451.878,E2 12451.878} C_VEL
LIN {X 0,Y 343.466,Z 980.825,A -85,B 0,C 180,E1 12449.994,E2 12449.994} C_VEL
LIN {X 0,Y 352.013,Z 960.399,A -85,B 0,C 180,E1 12448.461,E2 12448.461} C_VEL
LIN {X 0,Y 360.088,Z 938.623,A -85,B 0,C 180,E1 12447.113,E2 12447.113} C_VEL
LIN {X 0,Y 366.798,Z 917.2,A -85,B 0,C 180,E1 12446.057,E2 12446.057} C_VEL
LIN {X 0,Y 373.017,Z 893.881,A -85,B 0,C 180,E1 12445.141,E2 12445.141} C_VEL
LIN {X 0,Y 377.851,Z 870.545,A -85,B 0,C 180,E1 12444.451,E2 12444.451} C_VEL
LIN {X 0,Y 381.633,Z 846.025,A -85,B 0,C 180,E1 12443.897,E2 12443.897} C_VEL
LIN {X 0,Y 388.06,Z 774.584,A -85,B 0,C 180,E1 12442.684,E2 12442.684} C_VEL
LIN {X 0,Y 399.768,Z 641.005,A -85,B 0,C 180,E1 12440.497,E2 12440.497} C_VEL
LIN {X 0,Y 393.8,Z 629.694,A -85,B 0,C 180,E1 12437.663,E2 12437.663} C_VEL
LIN {X 0,Y 388.461,Z 620.129,A -85,B 0,C 180,E1 12434.687,E2 12434.687} C_VEL
LIN {X 0,Y 383.847,Z 612.442,A -85,B 0,C 180,E1 12431.571,E2 12431.571} C_VEL
LIN {X 0,Y 380.763,Z 607.708,A -85,B 0,C 180,E1 12428.989,E2 12428.989} C_VEL
LIN {X 0,Y 378.23,Z 603.684,A -85,B 0,C 180,E1 12426.222,E2 12426.222} C_VEL
LIN {X 0,Y 375.556,Z 600.008,A -85,B 0,C 180,E1 12421.373,E2 12421.373} C_VEL
LIN {X 0,Y 375.028,Z 599.554,A -85,B 0,C 180,E1 12418.472,E2 12418.472} C_VEL
LIN {X 0,Y 375.603,Z 601.604,A -85,B 0,C 180,E1 12414.347,E2 12414.347} C_VEL
LIN {X 0,Y 376.783,Z 603.511,A -85,B 0,C 180,E1 12411.915,E2 12411.915} C_VEL
LIN {X 0,Y 379.253,Z 608.369,A -85,B 0,C 180,E1 12408.595,E2 12408.595} C_VEL
LIN {X 0,Y 381.202,Z 612.09,A -85,B 0,C 180,E1 12406.654,E2 12406.654} C_VEL
LIN {X 0,Y 384.299,Z 617.729,A -85,B 0,C 180,E1 12404.145,E2 12404.145} C_VEL
LIN {X 0,Y 389.09,Z 627.023,A -85,B 0,C 180,E1 12400.99,E2 12400.99} C_VEL
LIN {X 0,Y 394.479,Z 638.166,A -85,B 0,C 180,E1 12398.045,E2 12398.045} C_VEL
LIN {X 0,Y 398.562,Z 646.896,A -85,B 0,C 180,E1 12396.096,E2 12396.096} C_VEL
LIN {X 0,Y 381.716,Z 845.726,A -85,B 0,C 180,E1 12392.901,E2 12392.901} C_VEL
LIN {X 0,Y 378.049,Z 870.56,A -85,B 0,C 180,E1 12392.369,E2 12392.369} C_VEL
LIN {X 0,Y 373.486,Z 892.922,A -85,B 0,C 180,E1 12391.727,E2 12391.727} C_VEL
LIN {X 0,Y 367.506,Z 915.707,A -85,B 0,C 180,E1 12390.852,E2 12390.852} C_VEL
LIN {X 0,Y 360.868,Z 936.924,A -85,B 0,C 180,E1 12389.825,E2 12389.825} C_VEL
LIN {X 0,Y 352.906,Z 958.27,A -85,B 0,C 180,E1 12388.521,E2 12388.521} C_VEL
LIN {X 0,Y 344.451,Z 978.291,A -85,B 0,C 180,E1 12387.027,E2 12387.027} C_VEL
LIN {X 0,Y 335.27,Z 997.271,A -85,B 0,C 180,E1 12385.276,E2 12385.276} C_VEL
LIN {X 0,Y 325.433,Z 1015.904,A -85,B 0,C 180,E1 12383.192,E2 12383.192} C_VEL
LIN {X 0,Y 315.354,Z 1033.001,A -85,B 0,C 180,E1 12380.827,E2 12380.827} C_VEL
LIN {X 0,Y 305.042,Z 1049.379,A -85,B 0,C 180,E1 12378.08,E2 12378.08} C_VEL
LIN {X 0,Y 295.187,Z 1063.855,A -85,B 0,C 180,E1 12375.069,E2 12375.069} C_VEL
LIN {X 0,Y 285.221,Z 1077.903,A -85,B 0,C 180,E1 12371.497,E2 12371.497} C_VEL
LIN {X 0,Y 276.352,Z 1089.849,A -85,B 0,C 180,E1 12367.696,E2 12367.696} C_VEL
LIN {X 0,Y 267.642,Z 1101.495,A -85,B 0,C 180,E1 12363.055,E2 12363.055} C_VEL
LIN {X 0,Y 261.414,Z 1109.926,A -85,B 0,C 180,E1 12358.812,E2 12358.812} C_VEL
LIN {X 0,Y 255.62,Z 1118.165,A -85,B 0,C 180,E1 12353.515,E2 12353.515} C_VEL
LIN {X 0,Y 252.041,Z 1123.819,A -85,B 0,C 180,E1 12348.744,E2 12348.744} C_VEL
LIN {X 0,Y 249.469,Z 1128.657,A -85,B 0,C 180,E1 12343.102,E2 12343.102} C_VEL
LIN {X 0,Y 248.428,Z 1131.357,A -85,B 0,C 180,E1 12338.331,E2 12338.331} C_VEL
LIN {X 0,Y 248.048,Z 1132.963,A -85,B 0,C 180,E1 12333.235,E2 12333.235} C_VEL
LIN {X 0,Y 248.018,Z 1133.147,A -85,B 0,C 180,E1 12328.614,E2 12328.614} C_VEL
LIN {X 0,Y 248.146,Z 1132.399,A -85,B 0,C 180,E1 12324.43,E2 12324.43} C_VEL
LIN {X 0,Y 248.764,Z 1130.443,A -85,B 0,C 180,E1 12319.579,E2 12319.579} C_VEL
LIN {X 0,Y 250.463,Z 1126.664,A -85,B 0,C 180,E1 12314.179,E2 12314.179} C_VEL
LIN {X 0,Y 253.52,Z 1121.5,A -85,B 0,C 180,E1 12308.967,E2 12308.967} C_VEL
LIN {X 0,Y 258.201,Z 1114.479,A -85,B 0,C 180,E1 12303.802,E2 12303.802} C_VEL
LIN {X 0,Y 264.271,Z 1106.2,A -85,B 0,C 180,E1 12299.031,E2 12299.031} C_VEL
LIN {X 0,Y 271.864,Z 1095.957,A -85,B 0,C 180,E1 12294.471,E2 12294.471} C_VEL
LIN {X 0,Y 280.539,Z 1084.439,A -85,B 0,C 180,E1 12290.342,E2 12290.342} C_VEL
LIN {X 0,Y 289.667,Z 1071.848,A -85,B 0,C 180,E1 12286.748,E2 12286.748} C_VEL
LIN {X 0,Y 299.859,Z 1057.325,A -85,B 0,C 180,E1 12283.37,E2 12283.37} C_VEL
LIN {X 0,Y 309.509,Z 1042.63,A -85,B 0,C 180,E1 12280.607,E2 12280.607} C_VEL
LIN {X 0,Y 320.137,Z 1025.363,A -85,B 0,C 180,E1 12277.941,E2 12277.941} C_VEL
LIN {X 0,Y 329.417,Z 1008.842,A -85,B 0,C 180,E1 12275.861,E2 12275.861} C_VEL
LIN {X 0,Y 339.109,Z 990.026,A -85,B 0,C 180,E1 12273.898,E2 12273.898} C_VEL
LIN {X 0,Y 347.772,Z 971.1,A -85,B 0,C 180,E1 12272.297,E2 12272.297} C_VEL
LIN {X 0,Y 356.333,Z 950.07,A -85,B 0,C 180,E1 12270.834,E2 12270.834} C_VEL
LIN {X 0,Y 363.26,Z 930.224,A -85,B 0,C 180,E1 12269.723,E2 12269.723} C_VEL
LIN {X 0,Y 369.962,Z 907.878,A -85,B 0,C 180,E1 12268.714,E2 12268.714} C_VEL
LIN {X 0,Y 375.176,Z 886.163,A -85,B 0,C 180,E1 12267.956,E2 12267.956} C_VEL
LIN {X 0,Y 379.689,Z 862.334,A -85,B 0,C 180,E1 12267.33,E2 12267.33} C_VEL
LIN {X 0,Y 382.543,Z 839.811,A -85,B 0,C 180,E1 12266.889,E2 12266.889} C_VEL
LIN {X 0,Y 398.758,Z 646.982,A -85,B 0,C 180,E1 12263.791,E2 12263.791} C_VEL
LIN {X 0,Y 394.342,Z 637.548,A -85,B 0,C 180,E1 12261.67,E2 12261.67} C_VEL
LIN {X 0,Y 392.451,Z 634.762,A -85,B 0,C 180,E1 12260.743,E2 12260.743} C_VEL
LIN {X 0,Y 389.056,Z 632.799,A -85,B 0,C 180,E1 12259.114,E2 12259.114} C_VEL
LIN {X 0,Y 385.942,Z 630.889,A -85,B 0,C 180,E1 12257.445,E2 12257.445} C_VEL
LIN {X 0,Y 384.879,Z 629.192,A -85,B 0,C 180,E1 12256.755,E2 12256.755} C_VEL
LIN {X 0,Y 381.315,Z 622.194,A -85,B 0,C 180,E1 12254.017,E2 12254.017} C_VEL
LIN {X 0,Y 378.629,Z 616.994,A -85,B 0,C 180,E1 12251.424,E2 12251.424} C_VEL
LIN {X 0,Y 376.918,Z 613.778,A -85,B 0,C 180,E1 12249.302,E2 12249.302} C_VEL
LIN {X 0,Y 375.543,Z 610.681,A -85,B 0,C 180,E1 12246.881,E2 12246.881} C_VEL
LIN {X 0,Y 374.359,Z 607.978,A -85,B 0,C 180,E1 12241.684,E2 12241.684} C_VEL
LIN {X 0,Y 374.84,Z 608.278,A -85,B 0,C 180,E1 12238.777,E2 12238.777} C_VEL
LIN {X 0,Y 377.538,Z 611.969,A -85,B 0,C 180,E1 12233.766,E2 12233.766} C_VEL
LIN {X 0,Y 380.754,Z 617.304,A -85,B 0,C 180,E1 12230.324,E2 12230.324} C_VEL
LIN {X 0,Y 383.569,Z 621.951,A -85,B 0,C 180,E1 12228.039,E2 12228.039} C_VEL
LIN {X 0,Y 387.38,Z 628.455,A -85,B 0,C 180,E1 12225.458,E2 12225.458} C_VEL
LIN {X 0,Y 392.5,Z 637.871,A -85,B 0,C 180,E1 12222.544,E2 12222.544} C_VEL
LIN {X 0,Y 396.585,Z 646.019,A -85,B 0,C 180,E1 12220.506,E2 12220.506} C_VEL
LIN {X 0,Y 378.712,Z 843.825,A -85,B 0,C 180,E1 12217.255,E2 12217.255} C_VEL
LIN {X 0,Y 374.82,Z 869.468,A -85,B 0,C 180,E1 12216.697,E2 12216.697} C_VEL
LIN {X 0,Y 370.16,Z 891.782,A -85,B 0,C 180,E1 12216.057,E2 12216.057} C_VEL
LIN {X 0,Y 364.065,Z 914.807,A -85,B 0,C 180,E1 12215.191,E2 12215.191} C_VEL
LIN {X 0,Y 357.579,Z 935.365,A -85,B 0,C 180,E1 12214.212,E2 12214.212} C_VEL
LIN {X 0,Y 348.97,Z 958.606,A -85,B 0,C 180,E1 12212.832,E2 12212.832} C_VEL
LIN {X 0,Y 340.795,Z 977.847,A -85,B 0,C 180,E1 12211.429,E2 12211.429} C_VEL
LIN {X 0,Y 330.633,Z 999.099,A -85,B 0,C 180,E1 12209.53,E2 12209.53} C_VEL
LIN {X 0,Y 321.581,Z 1016.198,A -85,B 0,C 180,E1 12207.67,E2 12207.67} C_VEL
LIN {X 0,Y 310.309,Z 1035.686,A -85,B 0,C 180,E1 12205.091,E2 12205.091} C_VEL
LIN {X 0,Y 300.741,Z 1050.974,A -85,B 0,C 180,E1 12202.619,E2 12202.619} C_VEL
LIN {X 0,Y 289.804,Z 1067.465,A -85,B 0,C 180,E1 12199.381,E2 12199.381} C_VEL
LIN {X 0,Y 280.307,Z 1081.031,A -85,B 0,C 180,E1 12196.101,E2 12196.101} C_VEL
LIN {X 0,Y 270.323,Z 1094.967,A -85,B 0,C 180,E1 12191.972,E2 12191.972} C_VEL
LIN {X 0,Y 262.231,Z 1106.078,A -85,B 0,C 180,E1 12187.872,E2 12187.872} C_VEL
LIN {X 0,Y 254.431,Z 1117.098,A -85,B 0,C 180,E1 12182.842,E2 12182.842} C_VEL
LIN {X 0,Y 248.84,Z 1125.387,A -85,B 0,C 180,E1 12178.043,E2 12178.043} C_VEL
LIN {X 0,Y 244.422,Z 1132.851,A -85,B 0,C 180,E1 12172.615,E2 12172.615} C_VEL
LIN {X 0,Y 241.733,Z 1138.274,A -85,B 0,C 180,E1 12167.327,E2 12167.327} C_VEL
LIN {X 0,Y 240.401,Z 1142.195,A -85,B 0,C 180,E1 12162.196,E2 12162.196} C_VEL
LIN {X 0,Y 239.987,Z 1144.84,A -85,B 0,C 180,E1 12156.699,E2 12156.699} C_VEL
LIN {X 0,Y 239.984,Z 1145.837,A -85,B 0,C 180,E1 12152.388,E2 12152.388} C_VEL
LIN {X 0,Y 240,Z 1145.905,A -85,B 0,C 180,E1 12148.329,E2 12148.329} C_VEL
LIN {X 0,Y 239.966,Z 1145.114,A -85,B 0,C 180,E1 12144.261,E2 12144.261} C_VEL
LIN {X 0,Y 240.166,Z 1143.229,A -85,B 0,C 180,E1 12139.687,E2 12139.687} C_VEL
LIN {X 0,Y 241.321,Z 1139.308,A -85,B 0,C 180,E1 12133.882,E2 12133.882} C_VEL
LIN {X 0,Y 243.54,Z 1134.384,A -85,B 0,C 180,E1 12128.82,E2 12128.82} C_VEL
LIN {X 0,Y 247.524,Z 1127.499,A -85,B 0,C 180,E1 12123.359,E2 12123.359} C_VEL
LIN {X 0,Y 253.166,Z 1118.798,A -85,B 0,C 180,E1 12118.12,E2 12118.12} C_VEL
LIN {X 0,Y 260.381,Z 1108.614,A -85,B 0,C 180,E1 12113.197,E2 12113.197} C_VEL
LIN {X 0,Y 268.66,Z 1097.078,A -85,B 0,C 180,E1 12108.795,E2 12108.795} C_VEL
LIN {X 0,Y 278.309,Z 1083.738,A -85,B 0,C 180,E1 12104.654,E2 12104.654} C_VEL
LIN {X 0,Y 287.592,Z 1070.432,A -85,B 0,C 180,E1 12101.324,E2 12101.324} C_VEL
LIN {X 0,Y 298.345,Z 1054.528,A -85,B 0,C 180,E1 12098.038,E2 12098.038} C_VEL
LIN {X 0,Y 308.703,Z 1038.026,A -85,B 0,C 180,E1 12095.29,E2 12095.29} C_VEL
LIN {X 0,Y 319.442,Z 1019.829,A -85,B 0,C 180,E1 12092.787,E2 12092.787} C_VEL
LIN {X 0,Y 329.219,Z 1001.481,A -85,B 0,C 180,E1 12090.737,E2 12090.737} C_VEL
LIN {X 0,Y 338.701,Z 982.133,A -85,B 0,C 180,E1 12088.936,E2 12088.936} C_VEL
LIN {X 0,Y 347.347,Z 962.095,A -85,B 0,C 180,E1 12087.425,E2 12087.425} C_VEL
LIN {X 0,Y 355.283,Z 941.429,A -85,B 0,C 180,E1 12086.132,E2 12086.132} C_VEL
LIN {X 0,Y 362.5,Z 919.352,A -85,B 0,C 180,E1 12085.027,E2 12085.027} C_VEL
LIN {X 0,Y 368.509,Z 897.718,A -85,B 0,C 180,E1 12084.166,E2 12084.166} C_VEL
LIN {X 0,Y 373.894,Z 873.267,A -85,B 0,C 180,E1 12083.419,E2 12083.419} C_VEL
LIN {X 0,Y 377.619,Z 850.794,A -85,B 0,C 180,E1 12082.897,E2 12082.897} C_VEL
LIN {X 0,Y 381.127,Z 816.472,A -85,B 0,C 180,E1 12082.289,E2 12082.289} C_VEL
LIN {X 0,Y 396.343,Z 645.698,A -85,B 0,C 180,E1 12079.49,E2 12079.49} C_VEL
LIN {X 0,Y 391.334,Z 635.973,A -85,B 0,C 180,E1 12076.973,E2 12076.973} C_VEL
LIN {X 0,Y 386.622,Z 627.279,A -85,B 0,C 180,E1 12074.223,E2 12074.223} C_VEL
LIN {X 0,Y 382.263,Z 619.856,A -85,B 0,C 180,E1 12071.161,E2 12071.161} C_VEL
LIN {X 0,Y 379.453,Z 615.398,A -85,B 0,C 180,E1 12068.715,E2 12068.715} C_VEL
LIN {X 0,Y 377.004,Z 611.431,A -85,B 0,C 180,E1 12065.937,E2 12065.937} C_VEL
LIN {X 0,Y 374.579,Z 607.967,A -85,B 0,C 180,E1 12061.377,E2 12061.377} C_VEL
LIN {X 0,Y 374.053,Z 607.499,A -85,B 0,C 180,E1 12058.468,E2 12058.468} C_VEL
LIN {X 0,Y 374.744,Z 609.771,A -85,B 0,C 180,E1 12054.027,E2 12054.027} C_VEL
LIN {X 0,Y 375.676,Z 611.325,A -85,B 0,C 180,E1 12052.122,E2 12052.122} C_VEL
LIN {X 0,Y 378.068,Z 616.199,A -85,B 0,C 180,E1 12048.791,E2 12048.791} C_VEL
LIN {X 0,Y 379.977,Z 619.985,A -85,B 0,C 180,E1 12046.835,E2 12046.835} C_VEL
LIN {X 0,Y 382.763,Z 625.211,A -85,B 0,C 180,E1 12044.508,E2 12044.508} C_VEL
LIN {X 0,Y 387.304,Z 634.319,A -85,B 0,C 180,E1 12041.407,E2 12041.407} C_VEL
LIN {X 0,Y 392.339,Z 645.06,A -85,B 0,C 180,E1 12038.548,E2 12038.548} C_VEL
LIN {X 0,Y 395.212,Z 651.516,A -85,B 0,C 180,E1 12037.098,E2 12037.098} C_VEL
LIN {X 0,Y 378.341,Z 845.672,A -85,B 0,C 180,E1 12033.997,E2 12033.997} C_VEL
LIN {X 0,Y 374.595,Z 870.564,A -85,B 0,C 180,E1 12033.471,E2 12033.471} C_VEL
LIN {X 0,Y 369.926,Z 893.01,A -85,B 0,C 180,E1 12032.835,E2 12032.835} C_VEL
LIN {X 0,Y 363.787,Z 915.92,A -85,B 0,C 180,E1 12031.965,E2 12031.965} C_VEL
LIN {X 0,Y 356.916,Z 937.417,A -85,B 0,C 180,E1 12030.935,E2 12030.935} C_VEL
LIN {X 0,Y 348.787,Z 958.671,A -85,B 0,C 180,E1 12029.644,E2 12029.644} C_VEL
LIN {X 0,Y 340.145,Z 978.653,A -85,B 0,C 180,E1 12028.163,E2 12028.163} C_VEL
LIN {X 0,Y 330.343,Z 998.367,A -85,B 0,C 180,E1 12026.344,E2 12026.344} C_VEL
LIN {X 0,Y 320.272,Z 1016.835,A -85,B 0,C 180,E1 12024.265,E2 12024.265} C_VEL
LIN {X 0,Y 309.99,Z 1033.776,A -85,B 0,C 180,E1 12021.91,E2 12021.91} C_VEL
LIN {X 0,Y 299.09,Z 1050.464,A -85,B 0,C 180,E1 12019.073,E2 12019.073} C_VEL
LIN {X 0,Y 289.496,Z 1064.102,A -85,B 0,C 180,E1 12016.209,E2 12016.209} C_VEL
LIN {X 0,Y 279.171,Z 1078.137,A -85,B 0,C 180,E1 12012.605,E2 12012.605} C_VEL
LIN {X 0,Y 270.373,Z 1089.516,A -85,B 0,C 180,E1 12008.954,E2 12008.954} C_VEL
LIN {X 0,Y 261.565,Z 1100.823,A -85,B 0,C 180,E1 12004.456,E2 12004.456} C_VEL
LIN {X 0,Y 254.585,Z 1109.754,A -85,B 0,C 180,E1 11999.921,E2 11999.921} C_VEL
LIN {X 0,Y 248.382,Z 1118.088,A -85,B 0,C 180,E1 11994.497,E2 11994.497} C_VEL
LIN {X 0,Y 244.503,Z 1123.79,A -85,B 0,C 180,E1 11989.593,E2 11989.593} C_VEL
LIN {X 0,Y 241.637,Z 1128.802,A -85,B 0,C 180,E1 11983.643,E2 11983.643} C_VEL
LIN {X 0,Y 240.501,Z 1131.46,A -85,B 0,C 180,E1 11978.849,E2 11978.849} C_VEL
LIN {X 0,Y 240.062,Z 1133.151,A -85,B 0,C 180,E1 11973.582,E2 11973.582} C_VEL
LIN {X 0,Y 240.021,Z 1133.379,A -85,B 0,C 180,E1 11968.806,E2 11968.806} C_VEL
LIN {X 0,Y 240.159,Z 1132.615,A -85,B 0,C 180,E1 11964.265,E2 11964.265} C_VEL
LIN {X 0,Y 240.829,Z 1130.654,A -85,B 0,C 180,E1 11959.232,E2 11959.232} C_VEL
LIN {X 0,Y 242.637,Z 1126.936,A -85,B 0,C 180,E1 11953.726,E2 11953.726} C_VEL
LIN {X 0,Y 245.76,Z 1121.96,A -85,B 0,C 180,E1 11948.52,E2 11948.52} C_VEL
LIN {X 0,Y 250.652,Z 1115.039,A -85,B 0,C 180,E1 11943.206,E2 11943.206} C_VEL
LIN {X 0,Y 256.651,Z 1107.209,A -85,B 0,C 180,E1 11938.53,E2 11938.53} C_VEL
LIN {X 0,Y 264.473,Z 1097.189,A -85,B 0,C 180,E1 11933.858,E2 11933.858} C_VEL
LIN {X 0,Y 272.909,Z 1086.448,A -85,B 0,C 180,E1 11929.847,E2 11929.847} C_VEL
LIN {X 0,Y 282.509,Z 1073.807,A -85,B 0,C 180,E1 11926.075,E2 11926.075} C_VEL
LIN {X 0,Y 292.089,Z 1060.72,A -85,B 0,C 180,E1 11922.897,E2 11922.897} C_VEL
LIN {X 0,Y 303.084,Z 1044.713,A -85,B 0,C 180,E1 11919.764,E2 11919.764} C_VEL
LIN {X 0,Y 313.308,Z 1028.802,A -85,B 0,C 180,E1 11917.226,E2 11917.226} C_VEL
LIN {X 0,Y 323.749,Z 1010.94,A -85,B 0,C 180,E1 11914.916,E2 11914.916} C_VEL
LIN {X 0,Y 333.292,Z 993.116,A -85,B 0,C 180,E1 11913.016,E2 11913.016} C_VEL
LIN {X 0,Y 342.829,Z 973.068,A -85,B 0,C 180,E1 11911.288,E2 11911.288} C_VEL
LIN {X 0,Y 351.561,Z 952.444,A -85,B 0,C 180,E1 11909.834,E2 11909.834} C_VEL
LIN {X 0,Y 358.986,Z 931.827,A -85,B 0,C 180,E1 11908.672,E2 11908.672} C_VEL
LIN {X 0,Y 365.813,Z 909.902,A -85,B 0,C 180,E1 11907.674,E2 11907.674} C_VEL
LIN {X 0,Y 371.434,Z 887.222,A -85,B 0,C 180,E1 11906.88,E2 11906.88} C_VEL
LIN {X 0,Y 376.059,Z 863.782,A -85,B 0,C 180,E1 11906.261,E2 11906.261} C_VEL
LIN {X 0,Y 379.126,Z 840.362,A -85,B 0,C 180,E1 11905.804,E2 11905.804} C_VEL
LIN {X 0,Y 395.454,Z 651.501,A -85,B 0,C 180,E1 11902.798,E2 11902.798} C_VEL
LIN {X 0,Y 390.232,Z 640.19,A -85,B 0,C 180,E1 11900.081,E2 11900.081} C_VEL
LIN {X 0,Y 386.123,Z 631.762,A -85,B 0,C 180,E1 11897.598,E2 11897.598} C_VEL
LIN {X 0,Y 384.879,Z 629.192,A -85,B 0,C 180,E1 11896.755,E2 11896.755} C_VEL
LIN {X 0,Y 383.405,Z 627.143,A -85,B 0,C 180,E1 11895.754,E2 11895.754} C_VEL
LIN {X 0,Y 380.944,Z 626.452,A -85,B 0,C 180,E1 11894.126,E2 11894.126} C_VEL
LIN {X 0,Y 378.318,Z 626.031,A -85,B 0,C 180,E1 11892.118,E2 11892.118} C_VEL
LIN {X 0,Y 377.727,Z 625.321,A -85,B 0,C 180,E1 11891.537,E2 11891.537} C_VEL
LIN {X 0,Y 375.74,Z 621.499,A -85,B 0,C 180,E1 11889.033,E2 11889.033} C_VEL
LIN {X 0,Y 374.424,Z 618.461,A -85,B 0,C 180,E1 11886.594,E2 11886.594} C_VEL
LIN {X 0,Y 373.391,Z 615.891,A -85,B 0,C 180,E1 11881.535,E2 11881.535} C_VEL
LIN {X 0,Y 373.909,Z 616.304,A -85,B 0,C 180,E1 11878.621,E2 11878.621} C_VEL
LIN {X 0,Y 376.536,Z 620.127,A -85,B 0,C 180,E1 11873.749,E2 11873.749} C_VEL
LIN {X 0,Y 379.427,Z 624.989,A -85,B 0,C 180,E1 11870.596,E2 11870.596} C_VEL
LIN {X 0,Y 382.162,Z 629.656,A -85,B 0,C 180,E1 11868.301,E2 11868.301} C_VEL
LIN {X 0,Y 385.943,Z 636.31,A -85,B 0,C 180,E1 11865.675,E2 11865.675} C_VEL
LIN {X 0,Y 390.709,Z 645.408,A -85,B 0,C 180,E1 11862.884,E2 11862.884} C_VEL
LIN {X 0,Y 393.312,Z 650.822,A -85,B 0,C 180,E1 11861.517,E2 11861.517} C_VEL
LIN {X 0,Y 375.483,Z 843.827,A -85,B 0,C 180,E1 11858.37,E2 11858.37} C_VEL
LIN {X 0,Y 371.524,Z 869.465,A -85,B 0,C 180,E1 11857.82,E2 11857.82} C_VEL
LIN {X 0,Y 366.785,Z 891.763,A -85,B 0,C 180,E1 11857.191,E2 11857.191} C_VEL
LIN {X 0,Y 360.344,Z 915.552,A -85,B 0,C 180,E1 11856.305,E2 11856.305} C_VEL
LIN {X 0,Y 353.625,Z 936.339,A -85,B 0,C 180,E1 11855.321,E2 11855.321} C_VEL
LIN {X 0,Y 344.947,Z 959.119,A -85,B 0,C 180,E1 11853.974,E2 11853.974} C_VEL
LIN {X 0,Y 336.59,Z 978.319,A -85,B 0,C 180,E1 11852.584,E2 11852.584} C_VEL
LIN {X 0,Y 326.197,Z 999.458,A -85,B 0,C 180,E1 11850.702,E2 11850.702} C_VEL
LIN {X 0,Y 316.743,Z 1016.831,A -85,B 0,C 180,E1 11848.814,E2 11848.814} C_VEL
LIN {X 0,Y 305.016,Z 1036.44,A -85,B 0,C 180,E1 11846.203,E2 11846.203} C_VEL
LIN {X 0,Y 295.184,Z 1051.65,A -85,B 0,C 180,E1 11843.726,E2 11843.726} C_VEL
LIN {X 0,Y 283.343,Z 1068.788,A -85,B 0,C 180,E1 11840.292,E2 11840.292} C_VEL
LIN {X 0,Y 273.584,Z 1082.218,A -85,B 0,C 180,E1 11836.967,E2 11836.967} C_VEL
LIN {X 0,Y 262.932,Z 1096.376,A -85,B 0,C 180,E1 11832.603,E2 11832.603} C_VEL
LIN {X 0,Y 254.555,Z 1107.43,A -85,B 0,C 180,E1 11828.362,E2 11828.362} C_VEL
LIN {X 0,Y 246.562,Z 1118.126,A -85,B 0,C 180,E1 11823.194,E2 11823.194} C_VEL
LIN {X 0,Y 240.851,Z 1126.258,A -85,B 0,C 180,E1 11818.247,E2 11818.247} C_VEL
LIN {X 0,Y 236.193,Z 1133.689,A -85,B 0,C 180,E1 11812.396,E2 11812.396} C_VEL
LIN {X 0,Y 233.647,Z 1138.703,A -85,B 0,C 180,E1 11807.175,E2 11807.175} C_VEL
LIN {X 0,Y 232.255,Z 1142.8,A -85,B 0,C 180,E1 11801.171,E2 11801.171} C_VEL
LIN {X 0,Y 231.978,Z 1144.845,A -85,B 0,C 180,E1 11796.186,E2 11796.186} C_VEL
LIN {X 0,Y 231.997,Z 1145.676,A -85,B 0,C 180,E1 11791.976,E2 11791.976} C_VEL
LIN {X 0,Y 231.997,Z 1145.671,A -85,B 0,C 180,E1 11788.024,E2 11788.024} C_VEL
LIN {X 0,Y 231.98,Z 1144.832,A -85,B 0,C 180,E1 11783.814,E2 11783.814} C_VEL
LIN {X 0,Y 232.286,Z 1142.658,A -85,B 0,C 180,E1 11778.579,E2 11778.579} C_VEL
LIN {X 0,Y 233.646,Z 1138.662,A -85,B 0,C 180,E1 11772.825,E2 11772.825} C_VEL
LIN {X 0,Y 236.037,Z 1133.901,A -85,B 0,C 180,E1 11767.851,E2 11767.851} C_VEL
LIN {X 0,Y 240.614,Z 1126.548,A -85,B 0,C 180,E1 11761.993,E2 11761.993} C_VEL
LIN {X 0,Y 246.249,Z 1118.457,A -85,B 0,C 180,E1 11757.036,E2 11757.036} C_VEL
LIN {X 0,Y 254.161,Z 1107.853,A -85,B 0,C 180,E1 11751.855,E2 11751.855} C_VEL
LIN {X 0,Y 262.471,Z 1096.843,A -85,B 0,C 180,E1 11747.601,E2 11747.601} C_VEL
LIN {X 0,Y 272.542,Z 1083.492,A -85,B 0,C 180,E1 11743.413,E2 11743.413} C_VEL
LIN {X 0,Y 282.759,Z 1069.396,A -85,B 0,C 180,E1 11739.883,E2 11739.883} C_VEL
LIN {X 0,Y 293.937,Z 1053.318,A -85,B 0,C 180,E1 11736.601,E2 11736.601} C_VEL
LIN {X 0,Y 304.27,Z 1037.348,A -85,B 0,C 180,E1 11733.963,E2 11733.963} C_VEL
LIN {X 0,Y 315.354,Z 1019.003,A -85,B 0,C 180,E1 11731.469,E2 11731.469} C_VEL
LIN {X 0,Y 325.288,Z 1000.808,A -85,B 0,C 180,E1 11729.46,E2 11729.46} C_VEL
LIN {X 0,Y 335.23,Z 980.894,A -85,B 0,C 180,E1 11727.642,E2 11727.642} C_VEL
LIN {X 0,Y 344.166,Z 960.493,A -85,B 0,C 180,E1 11726.139,E2 11726.139} C_VEL
LIN {X 0,Y 352.664,Z 938.545,A -85,B 0,C 180,E1 11724.811,E2 11724.811} C_VEL
LIN {X 0,Y 359.74,Z 916.811,A -85,B 0,C 180,E1 11723.768,E2 11723.768} C_VEL
LIN {X 0,Y 366.205,Z 893.331,A -85,B 0,C 180,E1 11722.876,E2 11722.876} C_VEL
LIN {X 0,Y 371.143,Z 870.27,A -85,B 0,C 180,E1 11722.217,E2 11722.217} C_VEL
LIN {X 0,Y 375.066,Z 845.517,A -85,B 0,C 180,E1 11721.677,E2 11721.677} C_VEL
LIN {X 0,Y 382.865,Z 762.032,A -85,B 0,C 180,E1 11720.285,E2 11720.285} C_VEL
LIN {X 0,Y 393.047,Z 650.35,A -85,B 0,C 180,E1 11718.465,E2 11718.465} C_VEL
LIN {X 0,Y 387.876,Z 640.186,A -85,B 0,C 180,E1 11715.666,E2 11715.666} C_VEL
LIN {X 0,Y 383.214,Z 631.559,A -85,B 0,C 180,E1 11712.661,E2 11712.661} C_VEL
LIN {X 0,Y 379.989,Z 626.156,A -85,B 0,C 180,E1 11710.154,E2 11710.154} C_VEL
LIN {X 0,Y 378.075,Z 622.982,A -85,B 0,C 180,E1 11708.364,E2 11708.364} C_VEL
LIN {X 0,Y 375.903,Z 619.305,A -85,B 0,C 180,E1 11705.801,E2 11705.801} C_VEL
LIN {X 0,Y 373.556,Z 615.854,A -85,B 0,C 180,E1 11701.227,E2 11701.227} C_VEL
LIN {X 0,Y 373.078,Z 615.445,A -85,B 0,C 180,E1 11698.464,E2 11698.464} C_VEL
LIN {X 0,Y 373.902,Z 617.945,A -85,B 0,C 180,E1 11693.705,E2 11693.705} C_VEL
LIN {X 0,Y 374.613,Z 619.254,A -85,B 0,C 180,E1 11692.253,E2 11692.253} C_VEL
LIN {X 0,Y 376.823,Z 623.896,A -85,B 0,C 180,E1 11689.063,E2 11689.063} C_VEL
LIN {X 0,Y 378.662,Z 627.681,A -85,B 0,C 180,E1 11687.107,E2 11687.107} C_VEL
LIN {X 0,Y 381.244,Z 632.69,A -85,B 0,C 180,E1 11684.873,E2 11684.873} C_VEL
LIN {X 0,Y 385.534,Z 641.613,A -85,B 0,C 180,E1 11681.828,E2 11681.828} C_VEL
LIN {X 0,Y 390.23,Z 651.954,A -85,B 0,C 180,E1 11679.057,E2 11679.057} C_VEL
LIN {X 0,Y 391.988,Z 656.008,A -85,B 0,C 180,E1 11678.121,E2 11678.121} C_VEL
LIN {X 0,Y 375.108,Z 845.608,A -85,B 0,C 180,E1 11675.114,E2 11675.114} C_VEL
LIN {X 0,Y 371.282,Z 870.567,A -85,B 0,C 180,E1 11674.593,E2 11674.593} C_VEL
LIN {X 0,Y 366.527,Z 893.008,A -85,B 0,C 180,E1 11673.967,E2 11673.967} C_VEL
LIN {X 0,Y 360.387,Z 915.544,A -85,B 0,C 180,E1 11673.126,E2 11673.126} C_VEL
LIN {X 0,Y 353.48,Z 936.785,A -85,B 0,C 180,E1 11672.126,E2 11672.126} C_VEL
LIN {X 0,Y 345.18,Z 958.178,A -85,B 0,C 180,E1 11670.852,E2 11670.852} C_VEL
LIN {X 0,Y 336.34,Z 978.224,A -85,B 0,C 180,E1 11669.389,E2 11669.389} C_VEL
LIN {X 0,Y 326.654,Z 997.363,A -85,B 0,C 180,E1 11667.655,E2 11667.655} C_VEL
LIN {X 0,Y 316.304,Z 1016.011,A -85,B 0,C 180,E1 11665.596,E2 11665.596} C_VEL
LIN {X 0,Y 305.448,Z 1033.449,A -85,B 0,C 180,E1 11663.198,E2 11663.198} C_VEL
LIN {X 0,Y 294.443,Z 1049.885,A -85,B 0,C 180,E1 11660.432,E2 11660.432} C_VEL
LIN {X 0,Y 283.925,Z 1064.35,A -85,B 0,C 180,E1 11657.395,E2 11657.395} C_VEL
LIN {X 0,Y 273.228,Z 1078.37,A -85,B 0,C 180,E1 11653.761,E2 11653.761} C_VEL
LIN {X 0,Y 264.077,Z 1089.746,A -85,B 0,C 180,E1 11650.067,E2 11650.067} C_VEL
LIN {X 0,Y 254.874,Z 1101.046,A -85,B 0,C 180,E1 11645.494,E2 11645.494} C_VEL
LIN {X 0,Y 247.543,Z 1109.974,A -85,B 0,C 180,E1 11640.863,E2 11640.863} C_VEL
LIN {X 0,Y 240.869,Z 1118.454,A -85,B 0,C 180,E1 11635.182,E2 11635.182} C_VEL
LIN {X 0,Y 236.698,Z 1124.253,A -85,B 0,C 180,E1 11630.009,E2 11630.009} C_VEL
LIN {X 0,Y 233.782,Z 1129.014,A -85,B 0,C 180,E1 11624.11,E2 11624.11} C_VEL
LIN {X 0,Y 232.548,Z 1131.672,A -85,B 0,C 180,E1 11619.154,E2 11619.154} C_VEL
LIN {X 0,Y 232.068,Z 1133.361,A -85,B 0,C 180,E1 11613.706,E2 11613.706} C_VEL
LIN {X 0,Y 232.023,Z 1133.588,A -85,B 0,C 180,E1 11608.765,E2 11608.765} C_VEL
LIN {X 0,Y 232.176,Z 1132.826,A -85,B 0,C 180,E1 11604.067,E2 11604.067} C_VEL
LIN {X 0,Y 232.906,Z 1130.865,A -85,B 0,C 180,E1 11598.861,E2 11598.861} C_VEL
LIN {X 0,Y 234.859,Z 1127.149,A -85,B 0,C 180,E1 11593.172,E2 11593.172} C_VEL
LIN {X 0,Y 238.203,Z 1122.174,A -85,B 0,C 180,E1 11587.803,E2 11587.803} C_VEL
LIN {X 0,Y 243.394,Z 1115.256,A -85,B 0,C 180,E1 11582.34,E2 11582.34} C_VEL
LIN {X 0,Y 249.721,Z 1107.427,A -85,B 0,C 180,E1 11577.551,E2 11577.551} C_VEL
LIN {X 0,Y 257.922,Z 1097.413,A -85,B 0,C 180,E1 11572.788,E2 11572.788} C_VEL
LIN {X 0,Y 266.724,Z 1086.673,A -85,B 0,C 180,E1 11568.716,E2 11568.716} C_VEL
LIN {X 0,Y 276.697,Z 1074.042,A -85,B 0,C 180,E1 11564.905,E2 11564.905} C_VEL
LIN {X 0,Y 286.615,Z 1060.961,A -85,B 0,C 180,E1 11561.706,E2 11561.706} C_VEL
LIN {X 0,Y 297.961,Z 1044.969,A -85,B 0,C 180,E1 11558.565,E2 11558.565} C_VEL
LIN {X 0,Y 308.15,Z 1029.568,A -85,B 0,C 180,E1 11556.103,E2 11556.103} C_VEL
LIN {X 0,Y 319.197,Z 1011.233,A -85,B 0,C 180,E1 11553.727,E2 11553.727} C_VEL
LIN {X 0,Y 328.973,Z 993.426,A -85,B 0,C 180,E1 11551.84,E2 11551.84} C_VEL
LIN {X 0,Y 338.817,Z 973.229,A -85,B 0,C 180,E1 11550.112,E2 11550.112} C_VEL
LIN {X 0,Y 347.346,Z 953.536,A -85,B 0,C 180,E1 11548.734,E2 11548.734} C_VEL
LIN {X 0,Y 355.219,Z 932.305,A -85,B 0,C 180,E1 11547.54,E2 11547.54} C_VEL
LIN {X 0,Y 362.174,Z 910.444,A -85,B 0,C 180,E1 11546.555,E2 11546.555} C_VEL
LIN {X 0,Y 367.985,Z 887.591,A -85,B 0,C 180,E1 11545.762,E2 11545.762} C_VEL
LIN {X 0,Y 372.708,Z 864.246,A -85,B 0,C 180,E1 11545.151,E2 11545.151} C_VEL
LIN {X 0,Y 375.887,Z 840.547,A -85,B 0,C 180,E1 11544.693,E2 11544.693} C_VEL
LIN {X 0,Y 392.23,Z 655.993,A -85,B 0,C 180,E1 11541.772,E2 11541.772} C_VEL
LIN {X 0,Y 387.539,Z 645.638,A -85,B 0,C 180,E1 11539.167,E2 11539.167} C_VEL
LIN {X 0,Y 384.031,Z 638.274,A -85,B 0,C 180,E1 11536.916,E2 11536.916} C_VEL
LIN {X 0,Y 380.185,Z 630.219,A -85,B 0,C 180,E1 11533.925,E2 11533.925} C_VEL
LIN {X 0,Y 377.727,Z 625.321,A -85,B 0,C 180,E1 11531.537,E2 11531.537} C_VEL
LIN {X 0,Y 376.527,Z 624.419,A -85,B 0,C 180,E1 11530.296,E2 11530.296} C_VEL
LIN {X 0,Y 373.491,Z 626.303,A -85,B 0,C 180,E1 11526.652,E2 11526.652} C_VEL
LIN {X 0,Y 373.237,Z 626.139,A -85,B 0,C 180,E1 11526.138,E2 11526.138} C_VEL
LIN {X 0,Y 372.424,Z 623.812,A -85,B 0,C 180,E1 11521.385,E2 11521.385} C_VEL
LIN {X 0,Y 372.98,Z 624.331,A -85,B 0,C 180,E1 11518.464,E2 11518.464} C_VEL
LIN {X 0,Y 375.372,Z 627.927,A -85,B 0,C 180,E1 11513.96,E2 11513.96} C_VEL
LIN {X 0,Y 378.108,Z 632.673,A -85,B 0,C 180,E1 11510.87,E2 11510.87} C_VEL
LIN {X 0,Y 380.764,Z 637.359,A -85,B 0,C 180,E1 11508.565,E2 11508.565} C_VEL
LIN {X 0,Y 384.628,Z 644.385,A -85,B 0,C 180,E1 11505.817,E2 11505.817} C_VEL
LIN {X 0,Y 389.381,Z 653.851,A -85,B 0,C 180,E1 11502.978,E2 11502.978} C_VEL
LIN {X 0,Y 390.153,Z 655.705,A -85,B 0,C 180,E1 11502.543,E2 11502.543} C_VEL
LIN {X 0,Y 372.386,Z 843.935,A -85,B 0,C 180,E1 11499.501,E2 11499.501} C_VEL
LIN {X 0,Y 368.364,Z 869.514,A -85,B 0,C 180,E1 11498.961,E2 11498.961} C_VEL
LIN {X 0,Y 363.536,Z 891.832,A -85,B 0,C 180,E1 11498.342,E2 11498.342} C_VEL
LIN {X 0,Y 356.943,Z 915.717,A -85,B 0,C 180,E1 11497.466,E2 11497.466} C_VEL
LIN {X 0,Y 350.028,Z 936.674,A -85,B 0,C 180,E1 11496.488,E2 11496.488} C_VEL
LIN {X 0,Y 341.452,Z 958.722,A -85,B 0,C 180,E1 11495.202,E2 11495.202} C_VEL
LIN {X 0,Y 333.046,Z 977.654,A -85,B 0,C 180,E1 11493.855,E2 11493.855} C_VEL
LIN {X 0,Y 322.186,Z 999.288,A -85,B 0,C 180,E1 11491.958,E2 11491.958} C_VEL
LIN {X 0,Y 312.568,Z 1016.531,A -85,B 0,C 180,E1 11490.103,E2 11490.103} C_VEL
LIN {X 0,Y 300.55,Z 1036.11,A -85,B 0,C 180,E1 11487.518,E2 11487.518} C_VEL
LIN {X 0,Y 290.375,Z 1051.387,A -85,B 0,C 180,E1 11485.039,E2 11485.039} C_VEL
LIN {X 0,Y 278.13,Z 1068.541,A -85,B 0,C 180,E1 11481.603,E2 11481.603} C_VEL
LIN {X 0,Y 267.996,Z 1081.976,A -85,B 0,C 180,E1 11478.262,E2 11478.262} C_VEL
LIN {X 0,Y 256.88,Z 1096.145,A -85,B 0,C 180,E1 11473.857,E2 11473.857} C_VEL
LIN {X 0,Y 248.099,Z 1107.202,A -85,B 0,C 180,E1 11469.552,E2 11469.552} C_VEL
LIN {X 0,Y 239.662,Z 1117.902,A -85,B 0,C 180,E1 11464.28,E2 11464.28} C_VEL
LIN {X 0,Y 233.517,Z 1126.148,A -85,B 0,C 180,E1 11459.131,E2 11459.131} C_VEL
LIN {X 0,Y 228.603,Z 1133.472,A -85,B 0,C 180,E1 11453.182,E2 11453.182} C_VEL
LIN {X 0,Y 225.842,Z 1138.488,A -85,B 0,C 180,E1 11447.788,E2 11447.788} C_VEL
LIN {X 0,Y 224.302,Z 1142.587,A -85,B 0,C 180,E1 11441.572,E2 11441.572} C_VEL
LIN {X 0,Y 223.983,Z 1144.634,A -85,B 0,C 180,E1 11436.408,E2 11436.408} C_VEL
LIN {X 0,Y 223.997,Z 1145.466,A -85,B 0,C 180,E1 11432.047,E2 11432.047} C_VEL
LIN {X 0,Y 223.997,Z 1145.461,A -85,B 0,C 180,E1 11427.953,E2 11427.953} C_VEL
LIN {X 0,Y 223.985,Z 1144.62,A -85,B 0,C 180,E1 11423.592,E2 11423.592} C_VEL
LIN {X 0,Y 224.337,Z 1142.444,A -85,B 0,C 180,E1 11418.169,E2 11418.169} C_VEL
LIN {X 0,Y 225.873,Z 1138.378,A -85,B 0,C 180,E1 11412.132,E2 11412.132} C_VEL
LIN {X 0,Y 228.599,Z 1133.419,A -85,B 0,C 180,E1 11406.818,E2 11406.818} C_VEL
LIN {X 0,Y 233.841,Z 1125.596,A -85,B 0,C 180,E1 11400.545,E2 11400.545} C_VEL
LIN {X 0,Y 239.981,Z 1117.4,A -85,B 0,C 180,E1 11395.483,E2 11395.483} C_VEL
LIN {X 0,Y 248.494,Z 1106.568,A -85,B 0,C 180,E1 11390.224,E2 11390.224} C_VEL
LIN {X 0,Y 257.231,Z 1095.574,A -85,B 0,C 180,E1 11385.982,E2 11385.982} C_VEL
LIN {X 0,Y 267.98,Z 1081.817,A -85,B 0,C 180,E1 11381.734,E2 11381.734} C_VEL
LIN {X 0,Y 278.113,Z 1068.362,A -85,B 0,C 180,E1 11378.393,E2 11378.393} C_VEL
LIN {X 0,Y 290.354,Z 1051.169,A -85,B 0,C 180,E1 11374.955,E2 11374.955} C_VEL
LIN {X 0,Y 300.826,Z 1035.411,A -85,B 0,C 180,E1 11372.408,E2 11372.408} C_VEL
LIN {X 0,Y 312.543,Z 1016.23,A -85,B 0,C 180,E1 11369.889,E2 11369.889} C_VEL
LIN {X 0,Y 322.241,Z 998.803,A -85,B 0,C 180,E1 11368.02,E2 11368.02} C_VEL
LIN {X 0,Y 333.022,Z 977.241,A -85,B 0,C 180,E1 11366.137,E2 11366.137} C_VEL
LIN {X 0,Y 341.428,Z 958.27,A -85,B 0,C 180,E1 11364.789,E2 11364.789} C_VEL
LIN {X 0,Y 350.396,Z 934.962,A -85,B 0,C 180,E1 11363.446,E2 11363.446} C_VEL
LIN {X 0,Y 357.141,Z 914.347,A -85,B 0,C 180,E1 11362.496,E2 11362.496} C_VEL
LIN {X 0,Y 363.875,Z 889.369,A -85,B 0,C 180,E1 11361.6,E2 11361.6} C_VEL
LIN {X 0,Y 368.58,Z 867.2,A -85,B 0,C 180,E1 11360.997,E2 11360.997} C_VEL
LIN {X 0,Y 372.383,Z 841.846,A -85,B 0,C 180,E1 11360.477,E2 11360.477} C_VEL
LIN {X 0,Y 389.933,Z 655.255,A -85,B 0,C 180,E1 11357.459,E2 11357.459} C_VEL
LIN {X 0,Y 384.663,Z 644.681,A -85,B 0,C 180,E1 11354.374,E2 11354.374} C_VEL
LIN {X 0,Y 380.692,Z 637.456,A -85,B 0,C 180,E1 11351.591,E2 11351.591} C_VEL
LIN {X 0,Y 377.996,Z 632.681,A -85,B 0,C 180,E1 11349.286,E2 11349.286} C_VEL
LIN {X 0,Y 375.035,Z 627.452,A -85,B 0,C 180,E1 11345.968,E2 11345.968} C_VEL
LIN {X 0,Y 372.536,Z 623.742,A -85,B 0,C 180,E1 11341.077,E2 11341.077} C_VEL
LIN {X 0,Y 372.1,Z 623.399,A -85,B 0,C 180,E1 11338.433,E2 11338.433} C_VEL
LIN {X 0,Y 373.001,Z 626.043,A -85,B 0,C 180,E1 11333.535,E2 11333.535} C_VEL
LIN {X 0,Y 373.628,Z 627.408,A -85,B 0,C 180,E1 11332.233,E2 11332.233} C_VEL
LIN {X 0,Y 375.587,Z 631.593,A -85,B 0,C 180,E1 11329.337,E2 11329.337} C_VEL
LIN {X 0,Y 377.671,Z 636.019,A -85,B 0,C 180,E1 11327.073,E2 11327.073} C_VEL
LIN {X 0,Y 379.919,Z 640.584,A -85,B 0,C 180,E1 11325.092,E2 11325.092} C_VEL
LIN {X 0,Y 383.838,Z 649.035,A -85,B 0,C 180,E1 11322.216,E2 11322.216} C_VEL
LIN {X 0,Y 388.153,Z 658.848,A -85,B 0,C 180,E1 11319.571,E2 11319.571} C_VEL
LIN {X 0,Y 388.867,Z 660.795,A -85,B 0,C 180,E1 11319.155,E2 11319.155} C_VEL
LIN {X 0,Y 372.009,Z 845.648,A -85,B 0,C 180,E1 11316.247,E2 11316.247} C_VEL
LIN {X 0,Y 368.114,Z 870.571,A -85,B 0,C 180,E1 11315.734,E2 11315.734} C_VEL
LIN {X 0,Y 363.27,Z 893.024,A -85,B 0,C 180,E1 11315.119,E2 11315.119} C_VEL
LIN {X 0,Y 356.849,Z 916.099,A -85,B 0,C 180,E1 11314.269,E2 11314.269} C_VEL
LIN {X 0,Y 349.425,Z 938.371,A -85,B 0,C 180,E1 11313.227,E2 11313.227} C_VEL
LIN {X 0,Y 340.966,Z 959.472,A -85,B 0,C 180,E1 11311.969,E2 11311.969} C_VEL
LIN {X 0,Y 331.616,Z 980,A -85,B 0,C 180,E1 11310.465,E2 11310.465} C_VEL
LIN {X 0,Y 321.695,Z 999.005,A -85,B 0,C 180,E1 11308.733,E2 11308.733} C_VEL
LIN {X 0,Y 310.879,Z 1017.773,A -85,B 0,C 180,E1 11306.633,E2 11306.633} C_VEL
LIN {X 0,Y 300.271,Z 1034.321,A -85,B 0,C 180,E1 11304.342,E2 11304.342} C_VEL
LIN {X 0,Y 288.714,Z 1050.969,A -85,B 0,C 180,E1 11301.508,E2 11301.508} C_VEL
LIN {X 0,Y 278.482,Z 1064.595,A -85,B 0,C 180,E1 11298.627,E2 11298.627} C_VEL
LIN {X 0,Y 267.401,Z 1078.604,A -85,B 0,C 180,E1 11294.969,E2 11294.969} C_VEL
LIN {X 0,Y 257.812,Z 1090.069,A -85,B 0,C 180,E1 11291.201,E2 11291.201} C_VEL
LIN {X 0,Y 248.27,Z 1101.269,A -85,B 0,C 180,E1 11286.588,E2 11286.588} C_VEL
LIN {X 0,Y 240.569,Z 1110.196,A -85,B 0,C 180,E1 11281.861,E2 11281.861} C_VEL
LIN {X 0,Y 233.64,Z 1118.523,A -85,B 0,C 180,E1 11276.155,E2 11276.155} C_VEL
LIN {X 0,Y 229.243,Z 1124.222,A -85,B 0,C 180,E1 11270.957,E2 11270.957} C_VEL
LIN {X 0,Y 225.94,Z 1129.228,A -85,B 0,C 180,E1 11264.611,E2 11264.611} C_VEL
LIN {X 0,Y 224.599,Z 1131.884,A -85,B 0,C 180,E1 11259.481,E2 11259.481} C_VEL
LIN {X 0,Y 224.075,Z 1133.571,A -85,B 0,C 180,E1 11253.838,E2 11253.838} C_VEL
LIN {X 0,Y 224.026,Z 1133.798,A -85,B 0,C 180,E1 11248.721,E2 11248.721} C_VEL
LIN {X 0,Y 224.179,Z 1133.089,A -85,B 0,C 180,E1 11244.064,E2 11244.064} C_VEL
LIN {X 0,Y 224.876,Z 1131.293,A -85,B 0,C 180,E1 11238.977,E2 11238.977} C_VEL
LIN {X 0,Y 226.98,Z 1127.561,A -85,B 0,C 180,E1 11232.834,E2 11232.834} C_VEL
LIN {X 0,Y 230.288,Z 1122.881,A -85,B 0,C 180,E1 11227.537,E2 11227.537} C_VEL
LIN {X 0,Y 236.195,Z 1115.473,A -85,B 0,C 180,E1 11221.421,E2 11221.421} C_VEL
LIN {X 0,Y 243.223,Z 1107.249,A -85,B 0,C 180,E1 11216.29,E2 11216.29} C_VEL
LIN {X 0,Y 251.928,Z 1097.095,A -85,B 0,C 180,E1 11211.434,E2 11211.434} C_VEL
LIN {X 0,Y 261.632,Z 1085.773,A -85,B 0,C 180,E1 11207.135,E2 11207.135} C_VEL
LIN {X 0,Y 272.106,Z 1072.899,A -85,B 0,C 180,E1 11203.316,E2 11203.316} C_VEL
LIN {X 0,Y 283.073,Z 1058.903,A -85,B 0,C 180,E1 11199.959,E2 11199.959} C_VEL
LIN {X 0,Y 294.251,Z 1043.399,A -85,B 0,C 180,E1 11197.008,E2 11197.008} C_VEL
LIN {X 0,Y 305.475,Z 1026.749,A -85,B 0,C 180,E1 11194.426,E2 11194.426} C_VEL
LIN {X 0,Y 316.189,Z 1009.119,A -85,B 0,C 180,E1 11192.229,E2 11192.229} C_VEL
LIN {X 0,Y 326.982,Z 989.567,A -85,B 0,C 180,E1 11190.246,E2 11190.246} C_VEL
LIN {X 0,Y 336.267,Z 970.563,A -85,B 0,C 180,E1 11188.695,E2 11188.695} C_VEL
LIN {X 0,Y 345.777,Z 948.361,A -85,B 0,C 180,E1 11187.226,E2 11187.226} C_VEL
LIN {X 0,Y 352.728,Z 929.522,A -85,B 0,C 180,E1 11186.226,E2 11186.226} C_VEL
LIN {X 0,Y 359.838,Z 906.897,A -85,B 0,C 180,E1 11185.26,E2 11185.26} C_VEL
LIN {X 0,Y 365.169,Z 885.848,A -85,B 0,C 180,E1 11184.563,E2 11184.563} C_VEL
LIN {X 0,Y 369.968,Z 861.624,A -85,B 0,C 180,E1 11183.959,E2 11183.959} C_VEL
LIN {X 0,Y 372.957,Z 839.208,A -85,B 0,C 180,E1 11183.537,E2 11183.537} C_VEL
LIN {X 0,Y 389.111,Z 660.678,A -85,B 0,C 180,E1 11180.731,E2 11180.731} C_VEL
LIN {X 0,Y 385.273,Z 651.936,A -85,B 0,C 180,E1 11178.459,E2 11178.459} C_VEL
LIN {X 0,Y 382.195,Z 645.212,A -85,B 0,C 180,E1 11176.373,E2 11176.373} C_VEL
LIN {X 0,Y 378.686,Z 637.634,A -85,B 0,C 180,E1 11173.514,E2 11173.514} C_VEL
LIN {X 0,Y 376.01,Z 632.135,A -85,B 0,C 180,E1 11170.728,E2 11170.728} C_VEL
LIN {X 0,Y 374.33,Z 628.707,A -85,B 0,C 180,E1 11168.371,E2 11168.371} C_VEL
LIN {X 0,Y 373.379,Z 626.344,A -85,B 0,C 180,E1 11166.458,E2 11166.458} C_VEL
LIN {X 0,Y 373.237,Z 626.139,A -85,B 0,C 180,E1 11166.138,E2 11166.138} C_VEL
LIN {X 0,Y 372.687,Z 626.411,A -85,B 0,C 180,E1 11164.948,E2 11164.948} C_VEL
LIN {X 0,Y 371.487,Z 631.452,A -85,B 0,C 180,E1 11161.411,E2 11161.411} C_VEL
LIN {X 0,Y 371.51,Z 631.713,A -85,B 0,C 180,E1 11160.722,E2 11160.722} C_VEL
LIN {X 0,Y 372.143,Z 632.582,A -85,B 0,C 180,E1 11157.998,E2 11157.998} C_VEL
LIN {X 0,Y 374.265,Z 635.843,A -85,B 0,C 180,E1 11154.096,E2 11154.096} C_VEL
LIN {X 0,Y 376.872,Z 640.503,A -85,B 0,C 180,E1 11151.071,E2 11151.071} C_VEL
LIN {X 0,Y 379.471,Z 645.23,A -85,B 0,C 180,E1 11148.756,E2 11148.756} C_VEL
LIN {X 0,Y 383.367,Z 652.6,A -85,B 0,C 180,E1 11145.924,E2 11145.924} C_VEL
LIN {X 0,Y 387.128,Z 660.559,A -85,B 0,C 180,E1 11143.585,E2 11143.585} C_VEL
LIN {X 0,Y 369.438,Z 844.051,A -85,B 0,C 180,E1 11140.652,E2 11140.652} C_VEL
LIN {X 0,Y 365.357,Z 869.537,A -85,B 0,C 180,E1 11140.122,E2 11140.122} C_VEL
LIN {X 0,Y 360.448,Z 891.86,A -85,B 0,C 180,E1 11139.514,E2 11139.514} C_VEL
LIN {X 0,Y 353.732,Z 915.754,A -85,B 0,C 180,E1 11138.654,E2 11138.654} C_VEL
LIN {X 0,Y 346.867,Z 936.192,A -85,B 0,C 180,E1 11137.718,E2 11137.718} C_VEL
LIN {X 0,Y 338.116,Z 958.328,A -85,B 0,C 180,E1 11136.455,E2 11136.455} C_VEL
LIN {X 0,Y 329.53,Z 977.29,A -85,B 0,C 180,E1 11135.129,E2 11135.129} C_VEL
LIN {X 0,Y 318.496,Z 998.825,A -85,B 0,C 180,E1 11133.274,E2 11133.274} C_VEL
LIN {X 0,Y 308.554,Z 1016.232,A -85,B 0,C 180,E1 11131.426,E2 11131.426} C_VEL
LIN {X 0,Y 296.168,Z 1035.898,A -85,B 0,C 180,E1 11128.853,E2 11128.853} C_VEL
LIN {X 0,Y 285.722,Z 1051.126,A -85,B 0,C 180,E1 11126.397,E2 11126.397} C_VEL
LIN {X 0,Y 273.067,Z 1068.295,A -85,B 0,C 180,E1 11122.964,E2 11122.964} C_VEL
LIN {X 0,Y 262.552,Z 1081.735,A -85,B 0,C 180,E1 11119.612,E2 11119.612} C_VEL
LIN {X 0,Y 250.87,Z 1096.02,A -85,B 0,C 180,E1 11115.132,E2 11115.132} C_VEL
LIN {X 0,Y 241.754,Z 1106.973,A -85,B 0,C 180,E1 11110.805,E2 11110.805} C_VEL
LIN {X 0,Y 232.852,Z 1117.68,A -85,B 0,C 180,E1 11105.43,E2 11105.43} C_VEL
LIN {X 0,Y 226.41,Z 1125.815,A -85,B 0,C 180,E1 11100.229,E2 11100.229} C_VEL
LIN {X 0,Y 221.002,Z 1133.331,A -85,B 0,C 180,E1 11093.947,E2 11093.947} C_VEL
LIN {X 0,Y 218.004,Z 1138.388,A -85,B 0,C 180,E1 11088.3,E2 11088.3} C_VEL
LIN {X 0,Y 216.356,Z 1142.375,A -85,B 0,C 180,E1 11082.003,E2 11082.003} C_VEL
LIN {X 0,Y 215.989,Z 1144.424,A -85,B 0,C 180,E1 11076.646,E2 11076.646} C_VEL
LIN {X 0,Y 215.997,Z 1145.256,A -85,B 0,C 180,E1 11072.122,E2 11072.122} C_VEL
LIN {X 0,Y 215.997,Z 1145.251,A -85,B 0,C 180,E1 11067.878,E2 11067.878} C_VEL
LIN {X 0,Y 215.99,Z 1144.409,A -85,B 0,C 180,E1 11063.354,E2 11063.354} C_VEL
LIN {X 0,Y 216.395,Z 1142.231,A -85,B 0,C 180,E1 11057.728,E2 11057.728} C_VEL
LIN {X 0,Y 218.06,Z 1138.228,A -85,B 0,C 180,E1 11051.555,E2 11051.555} C_VEL
LIN {X 0,Y 221.051,Z 1133.201,A -85,B 0,C 180,E1 11045.977,E2 11045.977} C_VEL
LIN {X 0,Y 226.675,Z 1125.374,A -85,B 0,C 180,E1 11039.517,E2 11039.517} C_VEL
LIN {X 0,Y 233.193,Z 1117.174,A -85,B 0,C 180,E1 11034.328,E2 11034.328} C_VEL
LIN {X 0,Y 242.168,Z 1106.335,A -85,B 0,C 180,E1 11028.966,E2 11028.966} C_VEL
LIN {X 0,Y 250.947,Z 1095.787,A -85,B 0,C 180,E1 11024.827,E2 11024.827} C_VEL
LIN {X 0,Y 262.745,Z 1081.306,A -85,B 0,C 180,E1 11020.312,E2 11020.312} C_VEL
LIN {X 0,Y 273.05,Z 1068.111,A -85,B 0,C 180,E1 11017.031,E2 11017.031} C_VEL
LIN {X 0,Y 285.702,Z 1050.901,A -85,B 0,C 180,E1 11013.597,E2 11013.597} C_VEL
LIN {X 0,Y 296.498,Z 1035.126,A -85,B 0,C 180,E1 11011.062,E2 11011.062} C_VEL
LIN {X 0,Y 308.53,Z 1015.923,A -85,B 0,C 180,E1 11008.566,E2 11008.566} C_VEL
LIN {X 0,Y 318.473,Z 998.479,A -85,B 0,C 180,E1 11006.718,E2 11006.718} C_VEL
LIN {X 0,Y 329.505,Z 976.867,A -85,B 0,C 180,E1 11004.861,E2 11004.861} C_VEL
LIN {X 0,Y 338.146,Z 957.741,A -85,B 0,C 180,E1 11003.528,E2 11003.528} C_VEL
LIN {X 0,Y 347.244,Z 934.467,A -85,B 0,C 180,E1 11002.216,E2 11002.216} C_VEL
LIN {X 0,Y 354.12,Z 913.788,A -85,B 0,C 180,E1 11001.284,E2 11001.284} C_VEL
LIN {X 0,Y 360.834,Z 889.206,A -85,B 0,C 180,E1 11000.423,E2 11000.423} C_VEL
LIN {X 0,Y 365.643,Z 866.871,A -85,B 0,C 180,E1 10999.829,E2 10999.829} C_VEL
LIN {X 0,Y 369.462,Z 841.706,A -85,B 0,C 180,E1 10999.322,E2 10999.322} C_VEL
LIN {X 0,Y 386.864,Z 660.136,A -85,B 0,C 180,E1 10996.401,E2 10996.401} C_VEL
LIN {X 0,Y 382.513,Z 651.214,A -85,B 0,C 180,E1 10993.684,E2 10993.684} C_VEL
LIN {X 0,Y 379.115,Z 644.818,A -85,B 0,C 180,E1 10991.178,E2 10991.178} C_VEL
LIN {X 0,Y 376.094,Z 639.18,A -85,B 0,C 180,E1 10988.408,E2 10988.408} C_VEL
LIN {X 0,Y 373.597,Z 634.927,A -85,B 0,C 180,E1 10985.375,E2 10985.375} C_VEL
LIN {X 0,Y 371.516,Z 631.63,A -85,B 0,C 180,E1 10980.925,E2 10980.925} C_VEL
LIN {X 0,Y 371.117,Z 631.384,A -85,B 0,C 180,E1 10978.302,E2 10978.302} C_VEL
LIN {X 0,Y 372.253,Z 634.35,A -85,B 0,C 180,E1 10973.057,E2 10973.057} C_VEL
LIN {X 0,Y 374.419,Z 639.421,A -85,B 0,C 180,E1 10969.537,E2 10969.537} C_VEL
LIN {X 0,Y 377.253,Z 645.387,A -85,B 0,C 180,E1 10966.512,E2 10966.512} C_VEL
LIN {X 0,Y 381.072,Z 653.946,A -85,B 0,C 180,E1 10963.381,E2 10963.381} C_VEL
LIN {X 0,Y 385.508,Z 664.229,A -85,B 0,C 180,E1 10960.452,E2 10960.452} C_VEL
LIN {X 0,Y 385.873,Z 665.568,A -85,B 0,C 180,E1 10960.207,E2 10960.207} C_VEL
LIN {X 0,Y 369.073,Z 845.54,A -85,B 0,C 180,E1 10957.401,E2 10957.401} C_VEL
LIN {X 0,Y 365.12,Z 870.444,A -85,B 0,C 180,E1 10956.898,E2 10956.898} C_VEL
LIN {X 0,Y 360.198,Z 892.889,A -85,B 0,C 180,E1 10956.296,E2 10956.296} C_VEL
LIN {X 0,Y 353.86,Z 915.374,A -85,B 0,C 180,E1 10955.487,E2 10955.487} C_VEL
LIN {X 0,Y 346.688,Z 936.642,A -85,B 0,C 180,E1 10954.52,E2 10954.52} C_VEL
LIN {X 0,Y 337.999,Z 958.206,A -85,B 0,C 180,E1 10953.278,E2 10953.278} C_VEL
LIN {X 0,Y 328.832,Z 978.155,A -85,B 0,C 180,E1 10951.862,E2 10951.862} C_VEL
LIN {X 0,Y 318.697,Z 997.34,A -85,B 0,C 180,E1 10950.17,E2 10950.17} C_VEL
LIN {X 0,Y 308.18,Z 1015.419,A -85,B 0,C 180,E1 10948.219,E2 10948.219} C_VEL
LIN {X 0,Y 296.991,Z 1032.591,A -85,B 0,C 180,E1 10945.916,E2 10945.916} C_VEL
LIN {X 0,Y 285.677,Z 1048.667,A -85,B 0,C 180,E1 10943.276,E2 10943.276} C_VEL
LIN {X 0,Y 274.379,Z 1063.322,A -85,B 0,C 180,E1 10940.258,E2 10940.258} C_VEL
LIN {X 0,Y 263.352,Z 1076.91,A -85,B 0,C 180,E1 10936.802,E2 10936.802} C_VEL
LIN {X 0,Y 252.802,Z 1089.082,A -85,B 0,C 180,E1 10932.867,E2 10932.867} C_VEL
LIN {X 0,Y 243.046,Z 1100.118,A -85,B 0,C 180,E1 10928.405,E2 10928.405} C_VEL
LIN {X 0,Y 234.376,Z 1109.627,A -85,B 0,C 180,E1 10923.39,E2 10923.39} C_VEL
LIN {X 0,Y 227.156,Z 1117.856,A -85,B 0,C 180,E1 10917.813,E2 10917.813} C_VEL
LIN {X 0,Y 222.042,Z 1123.944,A -85,B 0,C 180,E1 10912.226,E2 10912.226} C_VEL
LIN {X 0,Y 218.546,Z 1128.827,A -85,B 0,C 180,E1 10906.206,E2 10906.206} C_VEL
LIN {X 0,Y 216.76,Z 1131.877,A -85,B 0,C 180,E1 10900.364,E2 10900.364} C_VEL
LIN {X 0,Y 216.131,Z 1133.534,A -85,B 0,C 180,E1 10895.043,E2 10895.043} C_VEL
LIN {X 0,Y 216.027,Z 1134.074,A -85,B 0,C 180,E1 10889.47,E2 10889.47} C_VEL
LIN {X 0,Y 216.175,Z 1133.376,A -85,B 0,C 180,E1 10884.16,E2 10884.16} C_VEL
LIN {X 0,Y 216.847,Z 1131.722,A -85,B 0,C 180,E1 10879.102,E2 10879.102} C_VEL
LIN {X 0,Y 218.983,Z 1128.174,A -85,B 0,C 180,E1 10872.735,E2 10872.735} C_VEL
LIN {X 0,Y 222.58,Z 1123.342,A -85,B 0,C 180,E1 10866.994,E2 10866.994} C_VEL
LIN {X 0,Y 228.475,Z 1116.379,A -85,B 0,C 180,E1 10860.936,E2 10860.936} C_VEL
LIN {X 0,Y 235.357,Z 1108.654,A -85,B 0,C 180,E1 10855.889,E2 10855.889} C_VEL
LIN {X 0,Y 245.114,Z 1097.859,A -85,B 0,C 180,E1 10850.478,E2 10850.478} C_VEL
LIN {X 0,Y 254.685,Z 1087.125,A -85,B 0,C 180,E1 10846.292,E2 10846.292} C_VEL
LIN {X 0,Y 266.016,Z 1073.823,A -85,B 0,C 180,E1 10842.228,E2 10842.228} C_VEL
LIN {X 0,Y 277.303,Z 1059.921,A -85,B 0,C 180,E1 10838.845,E2 10838.845} C_VEL
LIN {X 0,Y 288.783,Z 1044.568,A -85,B 0,C 180,E1 10835.883,E2 10835.883} C_VEL
LIN {X 0,Y 300.284,Z 1028.093,A -85,B 0,C 180,E1 10833.302,E2 10833.302} C_VEL
LIN {X 0,Y 311.598,Z 1010.013,A -85,B 0,C 180,E1 10831.043,E2 10831.043} C_VEL
LIN {X 0,Y 322.101,Z 991.661,A -85,B 0,C 180,E1 10829.168,E2 10829.168} C_VEL
LIN {X 0,Y 332.102,Z 971.724,A -85,B 0,C 180,E1 10827.541,E2 10827.541} C_VEL
LIN {X 0,Y 341.409,Z 950.783,A -85,B 0,C 180,E1 10826.148,E2 10826.148} C_VEL
LIN {X 0,Y 349.307,Z 929.885,A -85,B 0,C 180,E1 10825.044,E2 10825.044} C_VEL
LIN {X 0,Y 356.578,Z 907.257,A -85,B 0,C 180,E1 10824.091,E2 10824.091} C_VEL
LIN {X 0,Y 362.057,Z 886.038,A -85,B 0,C 180,E1 10823.401,E2 10823.401} C_VEL
LIN {X 0,Y 366.913,Z 862.088,A -85,B 0,C 180,E1 10822.812,E2 10822.812} C_VEL
LIN {X 0,Y 369.994,Z 839.547,A -85,B 0,C 180,E1 10822.392,E2 10822.392} C_VEL
LIN {X 0,Y 386.121,Z 665.352,A -85,B 0,C 180,E1 10819.673,E2 10819.673} C_VEL
LIN {X 0,Y 381.76,Z 655.045,A -85,B 0,C 180,E1 10816.823,E2 10816.823} C_VEL
LIN {X 0,Y 377.77,Z 646.25,A -85,B 0,C 180,E1 10813.625,E2 10813.625} C_VEL
LIN {X 0,Y 374.842,Z 639.958,A -85,B 0,C 180,E1 10810.529,E2 10810.529} C_VEL
LIN {X 0,Y 373.212,Z 636.513,A -85,B 0,C 180,E1 10808.163,E2 10808.163} C_VEL
LIN {X 0,Y 372.336,Z 634.228,A -85,B 0,C 180,E1 10806.321,E2 10806.321} C_VEL
LIN {X 0,Y 371.449,Z 631.756,A -85,B 0,C 180,E1 10801.388,E2 10801.388} C_VEL
LIN {X 0,Y 371.51,Z 631.713,A -85,B 0,C 180,E1 10800.722,E2 10800.722} C_VEL
LIN {X 0,Y 371.588,Z 632.723,A -85,B 0,C 180,E1 10799.624,E2 10799.624} C_VEL
LIN {X 0,Y 371.61,Z 636.562,A -85,B 0,C 180,E1 10798.095,E2 10798.095} C_VEL
LIN {X 0,Y 371.957,Z 641.492,A -85,B 0,C 180,E1 10796.242,E2 10796.242} C_VEL
LIN {X 0,Y 372.335,Z 642.525,A -85,B 0,C 180,E1 10795.482,E2 10795.482} C_VEL
LIN {X 0,Y 373.211,Z 643.874,A -85,B 0,C 180,E1 10794.157,E2 10794.157} C_VEL
LIN {X 0,Y 375.569,Z 648.187,A -85,B 0,C 180,E1 10791.349,E2 10791.349} C_VEL
LIN {X 0,Y 378.003,Z 652.762,A -85,B 0,C 180,E1 10789.098,E2 10789.098} C_VEL
LIN {X 0,Y 381.669,Z 659.96,A -85,B 0,C 180,E1 10786.324,E2 10786.324} C_VEL
LIN {X 0,Y 384.215,Z 665.56,A -85,B 0,C 180,E1 10784.643,E2 10784.643} C_VEL
LIN {X 0,Y 366.654,Z 844.06,A -85,B 0,C 180,E1 10781.822,E2 10781.822} C_VEL
LIN {X 0,Y 362.503,Z 869.563,A -85,B 0,C 180,E1 10781.302,E2 10781.302} C_VEL
LIN {X 0,Y 357.513,Z 891.887,A -85,B 0,C 180,E1 10780.706,E2 10780.706} C_VEL
LIN {X 0,Y 350.865,Z 915.21,A -85,B 0,C 180,E1 10779.886,E2 10779.886} C_VEL
LIN {X 0,Y 343.869,Z 935.71,A -85,B 0,C 180,E1 10778.971,E2 10778.971} C_VEL
LIN {X 0,Y 334.544,Z 958.841,A -85,B 0,C 180,E1 10777.675,E2 10777.675} C_VEL
LIN {X 0,Y 325.787,Z 977.747,A -85,B 0,C 180,E1 10776.369,E2 10776.369} C_VEL
LIN {X 0,Y 314.513,Z 999.184,A -85,B 0,C 180,E1 10774.54,E2 10774.54} C_VEL
LIN {X 0,Y 303.972,Z 1017.163,A -85,B 0,C 180,E1 10772.641,E2 10772.641} C_VEL
LIN {X 0,Y 291.638,Z 1036.141,A -85,B 0,C 180,E1 10770.161,E2 10770.161} C_VEL
LIN {X 0,Y 280.563,Z 1051.803,A -85,B 0,C 180,E1 10767.634,E2 10767.634} C_VEL
LIN {X 0,Y 268.164,Z 1068.05,A -85,B 0,C 180,E1 10764.375,E2 10764.375} C_VEL
LIN {X 0,Y 257.26,Z 1081.496,A -85,B 0,C 180,E1 10761.018,E2 10761.018} C_VEL
LIN {X 0,Y 245.178,Z 1095.682,A -85,B 0,C 180,E1 10756.546,E2 10756.546} C_VEL
LIN {X 0,Y 235.529,Z 1106.745,A -85,B 0,C 180,E1 10752.126,E2 10752.126} C_VEL
LIN {X 0,Y 226.144,Z 1117.458,A -85,B 0,C 180,E1 10746.648,E2 10746.648} C_VEL
LIN {X 0,Y 219.301,Z 1125.595,A -85,B 0,C 180,E1 10741.317,E2 10741.317} C_VEL
LIN {X 0,Y 213.554,Z 1133.038,A -85,B 0,C 180,E1 10734.923,E2 10734.923} C_VEL
LIN {X 0,Y 210.308,Z 1138.056,A -85,B 0,C 180,E1 10729.151,E2 10729.151} C_VEL
LIN {X 0,Y 208.418,Z 1142.162,A -85,B 0,C 180,E1 10722.468,E2 10722.468} C_VEL
LIN {X 0,Y 207.997,Z 1144.213,A -85,B 0,C 180,E1 10716.903,E2 10716.903} C_VEL
LIN {X 0,Y 207.997,Z 1145.047,A -85,B 0,C 180,E1 10712.204,E2 10712.204} C_VEL
LIN {X 0,Y 208.003,Z 1145.066,A -85,B 0,C 180,E1 10708.072,E2 10708.072} C_VEL
LIN {X 0,Y 207.991,Z 1144.27,A -85,B 0,C 180,E1 10703.375,E2 10703.375} C_VEL
LIN {X 0,Y 208.337,Z 1142.376,A -85,B 0,C 180,E1 10698.09,E2 10698.09} C_VEL
LIN {X 0,Y 210.077,Z 1138.441,A -85,B 0,C 180,E1 10691.404,E2 10691.404} C_VEL
LIN {X 0,Y 213.171,Z 1133.509,A -85,B 0,C 180,E1 10685.621,E2 10685.621} C_VEL
LIN {X 0,Y 218.453,Z 1126.605,A -85,B 0,C 180,E1 10679.465,E2 10679.465} C_VEL
LIN {X 0,Y 225.437,Z 1118.167,A -85,B 0,C 180,E1 10673.827,E2 10673.827} C_VEL
LIN {X 0,Y 234.193,Z 1108.211,A -85,B 0,C 180,E1 10668.564,E2 10668.564} C_VEL
LIN {X 0,Y 244.141,Z 1096.724,A -85,B 0,C 180,E1 10663.878,E2 10663.878} C_VEL
LIN {X 0,Y 255.514,Z 1083.469,A -85,B 0,C 180,E1 10659.564,E2 10659.564} C_VEL
LIN {X 0,Y 266.892,Z 1069.427,A -85,B 0,C 180,E1 10655.979,E2 10655.979} C_VEL
LIN {X 0,Y 278.83,Z 1053.98,A -85,B 0,C 180,E1 10652.785,E2 10652.785} C_VEL
LIN {X 0,Y 290.557,Z 1037.426,A -85,B 0,C 180,E1 10650.061,E2 10650.061} C_VEL
LIN {X 0,Y 302.479,Z 1019.313,A -85,B 0,C 180,E1 10647.635,E2 10647.635} C_VEL
LIN {X 0,Y 313.348,Z 1000.856,A -85,B 0,C 180,E1 10645.65,E2 10645.65} C_VEL
LIN {X 0,Y 323.806,Z 981.402,A -85,B 0,C 180,E1 10643.931,E2 10643.931} C_VEL
LIN {X 0,Y 333.317,Z 961.091,A -85,B 0,C 180,E1 10642.49,E2 10642.49} C_VEL
LIN {X 0,Y 342.213,Z 939.637,A -85,B 0,C 180,E1 10641.24,E2 10641.24} C_VEL
LIN {X 0,Y 350.009,Z 917.106,A -85,B 0,C 180,E1 10640.207,E2 10640.207} C_VEL
LIN {X 0,Y 356.837,Z 893.676,A -85,B 0,C 180,E1 10639.363,E2 10639.363} C_VEL
LIN {X 0,Y 362.058,Z 870.53,A -85,B 0,C 180,E1 10638.736,E2 10638.736} C_VEL
LIN {X 0,Y 366.191,Z 845.844,A -85,B 0,C 180,E1 10638.224,E2 10638.224} C_VEL
LIN {X 0,Y 373.945,Z 768.07,A -85,B 0,C 180,E1 10636.967,E2 10636.967} C_VEL
LIN {X 0,Y 383.93,Z 665.078,A -85,B 0,C 180,E1 10635.328,E2 10635.328} C_VEL
LIN {X 0,Y 379.919,Z 656.685,A -85,B 0,C 180,E1 10632.618,E2 10632.618} C_VEL
LIN {X 0,Y 376.379,Z 649.896,A -85,B 0,C 180,E1 10629.712,E2 10629.712} C_VEL
LIN {X 0,Y 374.233,Z 646.045,A -85,B 0,C 180,E1 10627.523,E2 10627.523} C_VEL
LIN {X 0,Y 372.505,Z 642.801,A -85,B 0,C 180,E1 10625.236,E2 10625.236} C_VEL
LIN {X 0,Y 370.532,Z 639.587,A -85,B 0,C 180,E1 10620.928,E2 10620.928} C_VEL
LIN {X 0,Y 370.151,Z 639.289,A -85,B 0,C 180,E1 10618.452,E2 10618.452} C_VEL
LIN {X 0,Y 371.135,Z 642.129,A -85,B 0,C 180,E1 10613.347,E2 10613.347} C_VEL
LIN {X 0,Y 373.141,Z 646.985,A -85,B 0,C 180,E1 10609.891,E2 10609.891} C_VEL
LIN {X 0,Y 375.856,Z 652.944,A -85,B 0,C 180,E1 10606.853,E2 10606.853} C_VEL
LIN {X 0,Y 379.709,Z 661.85,A -85,B 0,C 180,E1 10603.595,E2 10603.595} C_VEL
LIN {X 0,Y 383.028,Z 670.17,A -85,B 0,C 180,E1 10601.276,E2 10601.276} C_VEL
LIN {X 0,Y 366.268,Z 845.622,A -85,B 0,C 180,E1 10598.571,E2 10598.571} C_VEL
LIN {X 0,Y 362.253,Z 870.443,A -85,B 0,C 180,E1 10598.078,E2 10598.078} C_VEL
LIN {X 0,Y 357.25,Z 892.882,A -85,B 0,C 180,E1 10597.488,E2 10597.488} C_VEL
LIN {X 0,Y 350.623,Z 915.928,A -85,B 0,C 180,E1 10596.674,E2 10596.674} C_VEL
LIN {X 0,Y 342.921,Z 938.24,A -85,B 0,C 180,E1 10595.671,E2 10595.671} C_VEL
LIN {X 0,Y 334.168,Z 959.287,A -85,B 0,C 180,E1 10594.462,E2 10594.462} C_VEL
LIN {X 0,Y 324.343,Z 980.03,A -85,B 0,C 180,E1 10592.992,E2 10592.992} C_VEL
LIN {X 0,Y 314.014,Z 998.979,A -85,B 0,C 180,E1 10591.313,E2 10591.313} C_VEL
LIN {X 0,Y 302.909,Z 1017.422,A -85,B 0,C 180,E1 10589.306,E2 10589.306} C_VEL
LIN {X 0,Y 291.831,Z 1033.865,A -85,B 0,C 180,E1 10587.081,E2 10587.081} C_VEL
LIN {X 0,Y 280.2,Z 1049.851,A -85,B 0,C 180,E1 10584.432,E2 10584.432} C_VEL
LIN {X 0,Y 268.63,Z 1064.327,A -85,B 0,C 180,E1 10581.413,E2 10581.413} C_VEL
LIN {X 0,Y 257.271,Z 1077.82,A -85,B 0,C 180,E1 10577.93,E2 10577.93} C_VEL
LIN {X 0,Y 246.368,Z 1089.873,A -85,B 0,C 180,E1 10573.949,E2 10573.949} C_VEL
LIN {X 0,Y 236.252,Z 1100.817,A -85,B 0,C 180,E1 10569.409,E2 10569.409} C_VEL
LIN {X 0,Y 227.23,Z 1110.244,A -85,B 0,C 180,E1 10564.281,E2 10564.281} C_VEL
LIN {X 0,Y 219.679,Z 1118.375,A -85,B 0,C 180,E1 10558.542,E2 10558.542} C_VEL
LIN {X 0,Y 214.328,Z 1124.407,A -85,B 0,C 180,E1 10552.781,E2 10552.781} C_VEL
LIN {X 0,Y 210.533,Z 1129.347,A -85,B 0,C 180,E1 10546.273,E2 10546.273} C_VEL
LIN {X 0,Y 208.779,Z 1132.198,A -85,B 0,C 180,E1 10540.486,E2 10540.486} C_VEL
LIN {X 0,Y 208.115,Z 1133.876,A -85,B 0,C 180,E1 10534.685,E2 10534.685} C_VEL
LIN {X 0,Y 208.031,Z 1134.261,A -85,B 0,C 180,E1 10529.174,E2 10529.174} C_VEL
LIN {X 0,Y 208.206,Z 1133.549,A -85,B 0,C 180,E1 10523.776,E2 10523.776} C_VEL
LIN {X 0,Y 208.988,Z 1131.825,A -85,B 0,C 180,E1 10518.408,E2 10518.408} C_VEL
LIN {X 0,Y 211.386,Z 1128.188,A -85,B 0,C 180,E1 10511.809,E2 10511.809} C_VEL
LIN {X 0,Y 215.328,Z 1123.308,A -85,B 0,C 180,E1 10505.881,E2 10505.881} C_VEL
LIN {X 0,Y 221.999,Z 1115.907,A -85,B 0,C 180,E1 10499.406,E2 10499.406} C_VEL
LIN {X 0,Y 229.416,Z 1108.081,A -85,B 0,C 180,E1 10494.265,E2 10494.265} C_VEL
LIN {X 0,Y 238.872,Z 1098.082,A -85,B 0,C 180,E1 10489.232,E2 10489.232} C_VEL
LIN {X 0,Y 248.849,Z 1087.349,A -85,B 0,C 180,E1 10484.994,E2 10484.994} C_VEL
LIN {X 0,Y 260.613,Z 1074.058,A -85,B 0,C 180,E1 10480.902,E2 10480.902} C_VEL
LIN {X 0,Y 272.279,Z 1060.16,A -85,B 0,C 180,E1 10477.512,E2 10477.512} C_VEL
LIN {X 0,Y 284.104,Z 1044.823,A -85,B 0,C 180,E1 10474.558,E2 10474.558} C_VEL
LIN {X 0,Y 295.917,Z 1028.358,A -85,B 0,C 180,E1 10471.992,E2 10471.992} C_VEL
LIN {X 0,Y 307.513,Z 1010.304,A -85,B 0,C 180,E1 10469.754,E2 10469.754} C_VEL
LIN {X 0,Y 318.418,Z 991.682,A -85,B 0,C 180,E1 10467.876,E2 10467.876} C_VEL
LIN {X 0,Y 328.616,Z 971.768,A -85,B 0,C 180,E1 10466.275,E2 10466.275} C_VEL
LIN {X 0,Y 337.955,Z 951.209,A -85,B 0,C 180,E1 10464.929,E2 10464.929} C_VEL
LIN {X 0,Y 345.998,Z 930.361,A -85,B 0,C 180,E1 10463.844,E2 10463.844} C_VEL
LIN {X 0,Y 353.207,Z 908.562,A -85,B 0,C 180,E1 10462.935,E2 10462.935} C_VEL
LIN {X 0,Y 358.993,Z 886.661,A -85,B 0,C 180,E1 10462.23,E2 10462.23} C_VEL
LIN {X 0,Y 363.931,Z 863.041,A -85,B 0,C 180,E1 10461.655,E2 10461.655} C_VEL
LIN {X 0,Y 367.176,Z 839.941,A -85,B 0,C 180,E1 10461.23,E2 10461.23} C_VEL
LIN {X 0,Y 383.27,Z 670.046,A -85,B 0,C 180,E1 10458.602,E2 10458.602} C_VEL
LIN {X 0,Y 379.381,Z 660.836,A -85,B 0,C 180,E1 10455.869,E2 10455.869} C_VEL
LIN {X 0,Y 375.984,Z 652.891,A -85,B 0,C 180,E1 10452.908,E2 10452.908} C_VEL
LIN {X 0,Y 373.447,Z 647.276,A -85,B 0,C 180,E1 10450.023,E2 10450.023} C_VEL
LIN {X 0,Y 371.361,Z 642.213,A -85,B 0,C 180,E1 10446.338,E2 10446.338} C_VEL
LIN {X 0,Y 370.474,Z 639.7,A -85,B 0,C 180,E1 10441.392,E2 10441.392} C_VEL
LIN {X 0,Y 370.966,Z 640.177,A -85,B 0,C 180,E1 10438.61,E2 10438.61} C_VEL
LIN {X 0,Y 372.335,Z 642.525,A -85,B 0,C 180,E1 10435.482,E2 10435.482} C_VEL
LIN {X 0,Y 372.879,Z 644.224,A -85,B 0,C 180,E1 10434.498,E2 10434.498} C_VEL
LIN {X 0,Y 373.521,Z 648.951,A -85,B 0,C 180,E1 10433.137,E2 10433.137} C_VEL
LIN {X 0,Y 374.596,Z 655.876,A -85,B 0,C 180,E1 10431.353,E2 10431.353} C_VEL
LIN {X 0,Y 375.341,Z 657.847,A -85,B 0,C 180,E1 10430.555,E2 10430.555} C_VEL
LIN {X 0,Y 378.748,Z 664.664,A -85,B 0,C 180,E1 10427.653,E2 10427.653} C_VEL
LIN {X 0,Y 381.424,Z 670.665,A -85,B 0,C 180,E1 10425.715,E2 10425.715} C_VEL
LIN {X 0,Y 364.011,Z 844.173,A -85,B 0,C 180,E1 10423.008,E2 10423.008} C_VEL
LIN {X 0,Y 359.792,Z 869.656,A -85,B 0,C 180,E1 10422.498,E2 10422.498} C_VEL
LIN {X 0,Y 354.717,Z 891.988,A -85,B 0,C 180,E1 10421.916,E2 10421.916} C_VEL
LIN {X 0,Y 347.738,Z 915.959,A -85,B 0,C 180,E1 10421.088,E2 10421.088} C_VEL
LIN {X 0,Y 340.623,Z 936.367,A -85,B 0,C 180,E1 10420.19,E2 10420.19} C_VEL
LIN {X 0,Y 331.404,Z 958.741,A -85,B 0,C 180,E1 10418.959,E2 10418.959} C_VEL
LIN {X 0,Y 322.201,Z 978.204,A -85,B 0,C 180,E1 10417.637,E2 10417.637} C_VEL
LIN {X 0,Y 311.08,Z 998.87,A -85,B 0,C 180,E1 10415.903,E2 10415.903} C_VEL
LIN {X 0,Y 300.665,Z 1016.251,A -85,B 0,C 180,E1 10414.103,E2 10414.103} C_VEL
LIN {X 0,Y 287.628,Z 1035.869,A -85,B 0,C 180,E1 10411.584,E2 10411.584} C_VEL
LIN {X 0,Y 276.125,Z 1051.683,A -85,B 0,C 180,E1 10409.056,E2 10409.056} C_VEL
LIN {X 0,Y 263.302,Z 1067.96,A -85,B 0,C 180,E1 10405.803,E2 10405.803} C_VEL
LIN {X 0,Y 252.127,Z 1081.255,A -85,B 0,C 180,E1 10402.482,E2 10402.482} C_VEL
LIN {X 0,Y 239.548,Z 1095.453,A -85,B 0,C 180,E1 10397.987,E2 10397.987} C_VEL
LIN {X 0,Y 229.437,Z 1106.516,A -85,B 0,C 180,E1 10393.517,E2 10393.517} C_VEL
LIN {X 0,Y 219.546,Z 1117.236,A -85,B 0,C 180,E1 10387.94,E2 10387.94} C_VEL
LIN {X 0,Y 212.275,Z 1125.374,A -85,B 0,C 180,E1 10382.478,E2 10382.478} C_VEL
LIN {X 0,Y 206.108,Z 1132.821,A -85,B 0,C 180,E1 10375.888,E2 10375.888} C_VEL
LIN {X 0,Y 202.584,Z 1137.841,A -85,B 0,C 180,E1 10369.911,E2 10369.911} C_VEL
LIN {X 0,Y 200.489,Z 1141.949,A -85,B 0,C 180,E1 10362.969,E2 10362.969} C_VEL
LIN {X 0,Y 199.998,Z 1144.001,A -85,B 0,C 180,E1 10357.18,E2 10357.18} C_VEL
LIN {X 0,Y 199.997,Z 1144.837,A -85,B 0,C 180,E1 10352.292,E2 10352.292} C_VEL
LIN {X 0,Y 200.003,Z 1144.856,A -85,B 0,C 180,E1 10347.994,E2 10347.994} C_VEL
LIN {X 0,Y 199.999,Z 1144.059,A -85,B 0,C 180,E1 10343.109,E2 10343.109} C_VEL
LIN {X 0,Y 200.399,Z 1142.163,A -85,B 0,C 180,E1 10337.611,E2 10337.611} C_VEL
LIN {X 0,Y 202.331,Z 1138.224,A -85,B 0,C 180,E1 10330.664,E2 10330.664} C_VEL
LIN {X 0,Y 205.695,Z 1133.29,A -85,B 0,C 180,E1 10324.674,E2 10324.674} C_VEL
LIN {X 0,Y 211.369,Z 1126.382,A -85,B 0,C 180,E1 10318.325,E2 10318.325} C_VEL
LIN {X 0,Y 218.768,Z 1117.973,A -85,B 0,C 180,E1 10312.563,E2 10312.563} C_VEL
LIN {X 0,Y 228.032,Z 1107.979,A -85,B 0,C 180,E1 10307.183,E2 10307.183} C_VEL
LIN {X 0,Y 238.462,Z 1096.489,A -85,B 0,C 180,E1 10302.44,E2 10302.44} C_VEL
LIN {X 0,Y 250.317,Z 1083.224,A -85,B 0,C 180,E1 10298.102,E2 10298.102} C_VEL
LIN {X 0,Y 262.115,Z 1069.177,A -85,B 0,C 180,E1 10294.515,E2 10294.515} C_VEL
LIN {X 0,Y 274.831,Z 1053.184,A -85,B 0,C 180,E1 10291.242,E2 10291.242} C_VEL
LIN {X 0,Y 286.519,Z 1037.149,A -85,B 0,C 180,E1 10288.635,E2 10288.635} C_VEL
LIN {X 0,Y 298.756,Z 1019.007,A -85,B 0,C 180,E1 10286.239,E2 10286.239} C_VEL
LIN {X 0,Y 309.829,Z 1000.634,A -85,B 0,C 180,E1 10284.293,E2 10284.293} C_VEL
LIN {X 0,Y 320.58,Z 981.036,A -85,B 0,C 180,E1 10282.597,E2 10282.597} C_VEL
LIN {X 0,Y 330.287,Z 960.686,A -85,B 0,C 180,E1 10281.184,E2 10281.184} C_VEL
LIN {X 0,Y 339.355,Z 939.166,A -85,B 0,C 180,E1 10279.962,E2 10279.962} C_VEL
LIN {X 0,Y 347.293,Z 916.544,A -85,B 0,C 180,E1 10278.952,E2 10278.952} C_VEL
LIN {X 0,Y 354.207,Z 893.028,A -85,B 0,C 180,E1 10278.13,E2 10278.13} C_VEL
LIN {X 0,Y 359.407,Z 870.267,A -85,B 0,C 180,E1 10277.531,E2 10277.531} C_VEL
LIN {X 0,Y 363.606,Z 845.379,A -85,B 0,C 180,E1 10277.027,E2 10277.027} C_VEL
LIN {X 0,Y 372.872,Z 753.796,A -85,B 0,C 180,E1 10275.572,E2 10275.572} C_VEL
LIN {X 0,Y 381.171,Z 670.235,A -85,B 0,C 180,E1 10274.275,E2 10274.275} C_VEL
LIN {X 0,Y 377.629,Z 662.705,A -85,B 0,C 180,E1 10271.687,E2 10271.687} C_VEL
LIN {X 0,Y 374.655,Z 656.881,A -85,B 0,C 180,E1 10269.06,E2 10269.06} C_VEL
LIN {X 0,Y 372.845,Z 653.516,A -85,B 0,C 180,E1 10267.086,E2 10267.086} C_VEL
LIN {X 0,Y 371.311,Z 650.558,A -85,B 0,C 180,E1 10264.943,E2 10264.943} C_VEL
LIN {X 0,Y 369.512,Z 647.475,A -85,B 0,C 180,E1 10260.775,E2 10260.775} C_VEL
LIN {X 0,Y 369.166,Z 647.285,A -85,B 0,C 180,E1 10258.293,E2 10258.293} C_VEL
LIN {X 0,Y 370.162,Z 650.161,A -85,B 0,C 180,E1 10253.33,E2 10253.33} C_VEL
LIN {X 0,Y 372.098,Z 655.075,A -85,B 0,C 180,E1 10249.941,E2 10249.941} C_VEL
LIN {X 0,Y 375.124,Z 662.081,A -85,B 0,C 180,E1 10246.552,E2 10246.552} C_VEL
LIN {X 0,Y 378.626,Z 670.641,A -85,B 0,C 180,E1 10243.586,E2 10243.586} C_VEL
LIN {X 0,Y 380.287,Z 675.104,A -85,B 0,C 180,E1 10242.357,E2 10242.357} C_VEL
LIN {X 0,Y 363.625,Z 845.652,A -85,B 0,C 180,E1 10239.758,E2 10239.758} C_VEL
LIN {X 0,Y 359.543,Z 870.442,A -85,B 0,C 180,E1 10239.275,E2 10239.275} C_VEL
LIN {X 0,Y 354.46,Z 892.876,A -85,B 0,C 180,E1 10238.7,E2 10238.7} C_VEL
LIN {X 0,Y 347.957,Z 915.203,A -85,B 0,C 180,E1 10237.932,E2 10237.932} C_VEL
LIN {X 0,Y 340.935,Z 935.373,A -85,B 0,C 180,E1 10237.058,E2 10237.058} C_VEL
LIN {X 0,Y 331.965,Z 957.094,A -85,B 0,C 180,E1 10235.874,E2 10235.874} C_VEL
LIN {X 0,Y 323.149,Z 975.669,A -85,B 0,C 180,E1 10234.624,E2 10234.624} C_VEL
LIN {X 0,Y 311.773,Z 996.65,A -85,B 0,C 180,E1 10232.871,E2 10232.871} C_VEL
LIN {X 0,Y 301.482,Z 1013.611,A -85,B 0,C 180,E1 10231.114,E2 10231.114} C_VEL
LIN {X 0,Y 288.954,Z 1032.131,A -85,B 0,C 180,E1 10228.729,E2 10228.729} C_VEL
LIN {X 0,Y 277.656,Z 1047.362,A -85,B 0,C 180,E1 10226.292,E2 10226.292} C_VEL
LIN {X 0,Y 264.757,Z 1063.258,A -85,B 0,C 180,E1 10223.095,E2 10223.095} C_VEL
LIN {X 0,Y 253.076,Z 1076.7,A -85,B 0,C 180,E1 10219.688,E2 10219.688} C_VEL
LIN {X 0,Y 241.065,Z 1089.574,A -85,B 0,C 180,E1 10215.494,E2 10215.494} C_VEL
LIN {X 0,Y 230.473,Z 1100.571,A -85,B 0,C 180,E1 10210.928,E2 10210.928} C_VEL
LIN {X 0,Y 220.921,Z 1110.068,A -85,B 0,C 180,E1 10205.722,E2 10205.722} C_VEL
LIN {X 0,Y 212.861,Z 1118.29,A -85,B 0,C 180,E1 10199.863,E2 10199.863} C_VEL
LIN {X 0,Y 207.068,Z 1124.377,A -85,B 0,C 180,E1 10193.93,E2 10193.93} C_VEL
LIN {X 0,Y 203.025,Z 1129.253,A -85,B 0,C 180,E1 10187.483,E2 10187.483} C_VEL
LIN {X 0,Y 200.916,Z 1132.301,A -85,B 0,C 180,E1 10181.192,E2 10181.192} C_VEL
LIN {X 0,Y 200.159,Z 1133.956,A -85,B 0,C 180,E1 10175.446,E2 10175.446} C_VEL
LIN {X 0,Y 200.035,Z 1134.515,A -85,B 0,C 180,E1 10169.714,E2 10169.714} C_VEL
LIN {X 0,Y 200.193,Z 1133.862,A -85,B 0,C 180,E1 10163.979,E2 10163.979} C_VEL
LIN {X 0,Y 200.955,Z 1132.253,A -85,B 0,C 180,E1 10158.52,E2 10158.52} C_VEL
LIN {X 0,Y 203.256,Z 1129,A -85,B 0,C 180,E1 10151.946,E2 10151.946} C_VEL
LIN {X 0,Y 207.456,Z 1124.015,A -85,B 0,C 180,E1 10145.512,E2 10145.512} C_VEL
LIN {X 0,Y 213.712,Z 1117.501,A -85,B 0,C 180,E1 10139.338,E2 10139.338} C_VEL
LIN {X 0,Y 221.615,Z 1109.487,A -85,B 0,C 180,E1 10133.768,E2 10133.768} C_VEL
LIN {X 0,Y 231.781,Z 1099.315,A -85,B 0,C 180,E1 10128.367,E2 10128.367} C_VEL
LIN {X 0,Y 242.051,Z 1088.701,A -85,B 0,C 180,E1 10124.046,E2 10124.046} C_VEL
LIN {X 0,Y 254.747,Z 1074.981,A -85,B 0,C 180,E1 10119.708,E2 10119.708} C_VEL
LIN {X 0,Y 266.093,Z 1061.919,A -85,B 0,C 180,E1 10116.472,E2 10116.472} C_VEL
LIN {X 0,Y 278.89,Z 1045.992,A -85,B 0,C 180,E1 10113.346,E2 10113.346} C_VEL
LIN {X 0,Y 290.254,Z 1030.626,A -85,B 0,C 180,E1 10110.932,E2 10110.932} C_VEL
LIN {X 0,Y 302.835,Z 1011.8,A -85,B 0,C 180,E1 10108.565,E2 10108.565} C_VEL
LIN {X 0,Y 313.565,Z 993.999,A -85,B 0,C 180,E1 10106.765,E2 10106.765} C_VEL
LIN {X 0,Y 324.192,Z 974.046,A -85,B 0,C 180,E1 10105.145,E2 10105.145} C_VEL
LIN {X 0,Y 332.896,Z 955.577,A -85,B 0,C 180,E1 10103.922,E2 10103.922} C_VEL
LIN {X 0,Y 342.021,Z 933.083,A -85,B 0,C 180,E1 10102.726,E2 10102.726} C_VEL
LIN {X 0,Y 348.69,Z 913.747,A -85,B 0,C 180,E1 10101.905,E2 10101.905} C_VEL
LIN {X 0,Y 355.53,Z 889.54,A -85,B 0,C 180,E1 10101.102,E2 10101.102} C_VEL
LIN {X 0,Y 360.372,Z 867.662,A -85,B 0,C 180,E1 10100.559,E2 10100.559} C_VEL
LIN {X 0,Y 364.191,Z 843.06,A -85,B 0,C 180,E1 10100.095,E2 10100.095} C_VEL
LIN {X 0,Y 380.546,Z 674.996,A -85,B 0,C 180,E1 10097.529,E2 10097.529} C_VEL
LIN {X 0,Y 377.514,Z 667.563,A -85,B 0,C 180,E1 10095.241,E2 10095.241} C_VEL
LIN {X 0,Y 374.457,Z 660.158,A -85,B 0,C 180,E1 10092.413,E2 10092.413} C_VEL
LIN {X 0,Y 372.178,Z 654.844,A -85,B 0,C 180,E1 10089.667,E2 10089.667} C_VEL
LIN {X 0,Y 370.255,Z 649.995,A -85,B 0,C 180,E1 10086.046,E2 10086.046} C_VEL
LIN {X 0,Y 369.509,Z 647.625,A -85,B 0,C 180,E1 10081.24,E2 10081.24} C_VEL
LIN {X 0,Y 370.027,Z 648.226,A -85,B 0,C 180,E1 10078.452,E2 10078.452} C_VEL
LIN {X 0,Y 372.008,Z 651.557,A -85,B 0,C 180,E1 10074.447,E2 10074.447} C_VEL
LIN {X 0,Y 374.342,Z 656.014,A -85,B 0,C 180,E1 10071.552,E2 10071.552} C_VEL
LIN {X 0,Y 375.341,Z 657.847,A -85,B 0,C 180,E1 10070.555,E2 10070.555} C_VEL
LIN {X 0,Y 375.895,Z 659.802,A -85,B 0,C 180,E1 10069.952,E2 10069.952} C_VEL
LIN {X 0,Y 376.447,Z 665.607,A -85,B 0,C 180,E1 10069.045,E2 10069.045} C_VEL
LIN {X 0,Y 377.015,Z 671.02,A -85,B 0,C 180,E1 10068.223,E2 10068.223} C_VEL
LIN {X 0,Y 377.557,Z 672.937,A -85,B 0,C 180,E1 10067.734,E2 10067.734} C_VEL
LIN {X 0,Y 378.748,Z 675.965,A -85,B 0,C 180,E1 10066.799,E2 10066.799} C_VEL
LIN {X 0,Y 361.54,Z 844.182,A -85,B 0,C 180,E1 10064.212,E2 10064.212} C_VEL
LIN {X 0,Y 357.267,Z 869.617,A -85,B 0,C 180,E1 10063.715,E2 10063.715} C_VEL
LIN {X 0,Y 352.127,Z 891.912,A -85,B 0,C 180,E1 10063.148,E2 10063.148} C_VEL
LIN {X 0,Y 345.199,Z 915.416,A -85,B 0,C 180,E1 10062.359,E2 10062.359} C_VEL
LIN {X 0,Y 337.958,Z 935.886,A -85,B 0,C 180,E1 10061.486,E2 10061.486} C_VEL
LIN {X 0,Y 328.702,Z 958.055,A -85,B 0,C 180,E1 10060.302,E2 10060.302} C_VEL
LIN {X 0,Y 319.594,Z 977.022,A -85,B 0,C 180,E1 10059.051,E2 10059.051} C_VEL
LIN {X 0,Y 307.827,Z 998.556,A -85,B 0,C 180,E1 10057.294,E2 10057.294} C_VEL
LIN {X 0,Y 296.783,Z 1016.568,A -85,B 0,C 180,E1 10055.458,E2 10055.458} C_VEL
LIN {X 0,Y 283.801,Z 1035.6,A -85,B 0,C 180,E1 10053.047,E2 10053.047} C_VEL
LIN {X 0,Y 272.081,Z 1051.281,A -85,B 0,C 180,E1 10050.572,E2 10050.572} C_VEL
LIN {X 0,Y 258.874,Z 1067.559,A -85,B 0,C 180,E1 10047.354,E2 10047.354} C_VEL
LIN {X 0,Y 247.165,Z 1081.015,A -85,B 0,C 180,E1 10044.007,E2 10044.007} C_VEL
LIN {X 0,Y 234.077,Z 1095.224,A -85,B 0,C 180,E1 10039.495,E2 10039.495} C_VEL
LIN {X 0,Y 223.486,Z 1106.289,A -85,B 0,C 180,E1 10034.984,E2 10034.984} C_VEL
LIN {X 0,Y 212.878,Z 1117.204,A -85,B 0,C 180,E1 10029.194,E2 10029.194} C_VEL
LIN {X 0,Y 205.112,Z 1125.404,A -85,B 0,C 180,E1 10023.529,E2 10023.529} C_VEL
LIN {X 0,Y 198.497,Z 1132.868,A -85,B 0,C 180,E1 10016.636,E2 10016.636} C_VEL
LIN {X 0,Y 194.754,Z 1137.84,A -85,B 0,C 180,E1 10010.434,E2 10010.434} C_VEL
LIN {X 0,Y 192.521,Z 1141.857,A -85,B 0,C 180,E1 10003.21,E2 10003.21} C_VEL
LIN {X 0,Y 191.995,Z 1143.79,A -85,B 0,C 180,E1 9997.481,E2 9997.481} C_VEL
LIN {X 0,Y 191.993,Z 1144.603,A -85,B 0,C 180,E1 9992.687,E2 9992.687} C_VEL
LIN {X 0,Y 192.01,Z 1144.67,A -85,B 0,C 180,E1 9988.209,E2 9988.209} C_VEL
LIN {X 0,Y 191.999,Z 1143.919,A -85,B 0,C 180,E1 9983.121,E2 9983.121} C_VEL
LIN {X 0,Y 192.379,Z 1142.188,A -85,B 0,C 180,E1 9977.696,E2 9977.696} C_VEL
LIN {X 0,Y 194.234,Z 1138.651,A -85,B 0,C 180,E1 9970.764,E2 9970.764} C_VEL
LIN {X 0,Y 198.061,Z 1133.335,A -85,B 0,C 180,E1 9963.946,E2 9963.946} C_VEL
LIN {X 0,Y 204.061,Z 1126.516,A -85,B 0,C 180,E1 9957.385,E2 9957.385} C_VEL
LIN {X 0,Y 211.841,Z 1118.164,A -85,B 0,C 180,E1 9951.461,E2 9951.461} C_VEL
LIN {X 0,Y 221.53,Z 1108.254,A -85,B 0,C 180,E1 9945.965,E2 9945.965} C_VEL
LIN {X 0,Y 232.388,Z 1096.84,A -85,B 0,C 180,E1 9941.152,E2 9941.152} C_VEL
LIN {X 0,Y 244.674,Z 1083.69,A -85,B 0,C 180,E1 9936.776,E2 9936.776} C_VEL
LIN {X 0,Y 256.85,Z 1069.711,A -85,B 0,C 180,E1 9933.178,E2 9933.178} C_VEL
LIN {X 0,Y 269.932,Z 1053.857,A -85,B 0,C 180,E1 9929.912,E2 9929.912} C_VEL
LIN {X 0,Y 282.291,Z 1037.385,A -85,B 0,C 180,E1 9927.245,E2 9927.245} C_VEL
LIN {X 0,Y 294.446,Z 1019.919,A -85,B 0,C 180,E1 9924.948,E2 9924.948} C_VEL
LIN {X 0,Y 306.211,Z 1000.884,A -85,B 0,C 180,E1 9922.951,E2 9922.951} C_VEL
LIN {X 0,Y 317.124,Z 981.464,A -85,B 0,C 180,E1 9921.296,E2 9921.296} C_VEL
LIN {X 0,Y 327.015,Z 961.189,A -85,B 0,C 180,E1 9919.911,E2 9919.911} C_VEL
LIN {X 0,Y 336.244,Z 939.766,A -85,B 0,C 180,E1 9918.715,E2 9918.715} C_VEL
LIN {X 0,Y 343.915,Z 918.49,A -85,B 0,C 180,E1 9917.775,E2 9917.775} C_VEL
LIN {X 0,Y 350.616,Z 896.617,A -85,B 0,C 180,E1 9917.007,E2 9917.007} C_VEL
LIN {X 0,Y 356.405,Z 872.496,A -85,B 0,C 180,E1 9916.366,E2 9916.366} C_VEL
LIN {X 0,Y 360.725,Z 848.552,A -85,B 0,C 180,E1 9915.877,E2 9915.877} C_VEL
LIN {X 0,Y 365.855,Z 800.845,A -85,B 0,C 180,E1 9915.115,E2 9915.115} C_VEL
LIN {X 0,Y 378.479,Z 675.38,A -85,B 0,C 180,E1 9913.171,E2 9913.171} C_VEL
LIN {X 0,Y 375.347,Z 668.58,A -85,B 0,C 180,E1 9910.669,E2 9910.669} C_VEL
LIN {X 0,Y 372.638,Z 663.12,A -85,B 0,C 180,E1 9908.021,E2 9908.021} C_VEL
LIN {X 0,Y 370.23,Z 658.432,A -85,B 0,C 180,E1 9904.803,E2 9904.803} C_VEL
LIN {X 0,Y 368.495,Z 655.365,A -85,B 0,C 180,E1 9900.622,E2 9900.622} C_VEL
LIN {X 0,Y 368.185,Z 655.283,A -85,B 0,C 180,E1 9898.132,E2 9898.132} C_VEL
LIN {X 0,Y 369.143,Z 658.202,A -85,B 0,C 180,E1 9893.389,E2 9893.389} C_VEL
LIN {X 0,Y 370.938,Z 662.9,A -85,B 0,C 180,E1 9890.144,E2 9890.144} C_VEL
LIN {X 0,Y 373.693,Z 669.559,A -85,B 0,C 180,E1 9886.933,E2 9886.933} C_VEL
LIN {X 0,Y 376.963,Z 677.927,A -85,B 0,C 180,E1 9884.026,E2 9884.026} C_VEL
LIN {X 0,Y 377.669,Z 680.149,A -85,B 0,C 180,E1 9883.451,E2 9883.451} C_VEL
LIN {X 0,Y 361.151,Z 845.576,A -85,B 0,C 180,E1 9880.964,E2 9880.964} C_VEL
LIN {X 0,Y 356.992,Z 870.443,A -85,B 0,C 180,E1 9880.491,E2 9880.491} C_VEL
LIN {X 0,Y 351.804,Z 892.975,A -85,B 0,C 180,E1 9879.927,E2 9879.927} C_VEL
LIN {X 0,Y 345.037,Z 915.756,A -85,B 0,C 180,E1 9879.161,E2 9879.161} C_VEL
LIN {X 0,Y 337.344,Z 937.358,A -85,B 0,C 180,E1 9878.238,E2 9878.238} C_VEL
LIN {X 0,Y 328.358,Z 958.386,A -85,B 0,C 180,E1 9877.095,E2 9877.095} C_VEL
LIN {X 0,Y 318.582,Z 978.449,A -85,B 0,C 180,E1 9875.749,E2 9875.749} C_VEL
LIN {X 0,Y 307.79,Z 997.63,A -85,B 0,C 180,E1 9874.141,E2 9874.141} C_VEL
LIN {X 0,Y 296.451,Z 1015.83,A -85,B 0,C 180,E1 9872.26,E2 9872.26} C_VEL
LIN {X 0,Y 284.098,Z 1033.404,A -85,B 0,C 180,E1 9869.975,E2 9869.975} C_VEL
LIN {X 0,Y 271.831,Z 1049.451,A -85,B 0,C 180,E1 9867.389,E2 9867.389} C_VEL
LIN {X 0,Y 259.471,Z 1064.056,A -85,B 0,C 180,E1 9864.401,E2 9864.401} C_VEL
LIN {X 0,Y 246.913,Z 1078.017,A -85,B 0,C 180,E1 9860.822,E2 9860.822} C_VEL
LIN {X 0,Y 234.892,Z 1090.334,A -85,B 0,C 180,E1 9856.712,E2 9856.712} C_VEL
LIN {X 0,Y 223.876,Z 1101.261,A -85,B 0,C 180,E1 9852.063,E2 9852.063} C_VEL
LIN {X 0,Y 213.931,Z 1110.685,A -85,B 0,C 180,E1 9846.745,E2 9846.745} C_VEL
LIN {X 0,Y 205.5,Z 1118.801,A -85,B 0,C 180,E1 9840.723,E2 9840.723} C_VEL
LIN {X 0,Y 199.42,Z 1124.839,A -85,B 0,C 180,E1 9834.593,E2 9834.593} C_VEL
LIN {X 0,Y 194.946,Z 1129.859,A -85,B 0,C 180,E1 9827.444,E2 9827.444} C_VEL
LIN {X 0,Y 192.884,Z 1132.731,A -85,B 0,C 180,E1 9821.058,E2 9821.058} C_VEL
LIN {X 0,Y 192.111,Z 1134.411,A -85,B 0,C 180,E1 9814.478,E2 9814.478} C_VEL
LIN {X 0,Y 192.038,Z 1134.643,A -85,B 0,C 180,E1 9808.591,E2 9808.591} C_VEL
LIN {X 0,Y 192.263,Z 1133.942,A -85,B 0,C 180,E1 9803.13,E2 9803.13} C_VEL
LIN {X 0,Y 193.281,Z 1132.138,A -85,B 0,C 180,E1 9797.147,E2 9797.147} C_VEL
LIN {X 0,Y 196.362,Z 1128.215,A -85,B 0,C 180,E1 9789.741,E2 9789.741} C_VEL
LIN {X 0,Y 201.078,Z 1123.243,A -85,B 0,C 180,E1 9783.414,E2 9783.414} C_VEL
LIN {X 0,Y 208.466,Z 1115.997,A -85,B 0,C 180,E1 9776.853,E2 9776.853} C_VEL
LIN {X 0,Y 217.24,Z 1107.723,A -85,B 0,C 180,E1 9771.247,E2 9771.247} C_VEL
LIN {X 0,Y 227.777,Z 1097.518,A -85,B 0,C 180,E1 9766.085,E2 9766.085} C_VEL
LIN {X 0,Y 239.336,Z 1086.093,A -85,B 0,C 180,E1 9761.598,E2 9761.598} C_VEL
LIN {X 0,Y 251.521,Z 1073.146,A -85,B 0,C 180,E1 9757.711,E2 9757.711} C_VEL
LIN {X 0,Y 264.162,Z 1058.927,A -85,B 0,C 180,E1 9754.332,E2 9754.332} C_VEL
LIN {X 0,Y 276.66,Z 1043.504,A -85,B 0,C 180,E1 9751.467,E2 9751.467} C_VEL
LIN {X 0,Y 289.431,Z 1026.376,A -85,B 0,C 180,E1 9748.925,E2 9748.925} C_VEL
LIN {X 0,Y 300.604,Z 1009.682,A -85,B 0,C 180,E1 9746.945,E2 9746.945} C_VEL
LIN {X 0,Y 312.407,Z 990.16,A -85,B 0,C 180,E1 9745.072,E2 9745.072} C_VEL
LIN {X 0,Y 322.484,Z 971.18,A -85,B 0,C 180,E1 9743.619,E2 9743.619} C_VEL
LIN {X 0,Y 332.342,Z 950.065,A -85,B 0,C 180,E1 9742.308,E2 9742.308} C_VEL
LIN {X 0,Y 340.268,Z 930.184,A -85,B 0,C 180,E1 9741.327,E2 9741.327} C_VEL
LIN {X 0,Y 347.874,Z 907.791,A -85,B 0,C 180,E1 9740.442,E2 9740.442} C_VEL
LIN {X 0,Y 353.729,Z 886.276,A -85,B 0,C 180,E1 9739.789,E2 9739.789} C_VEL
LIN {X 0,Y 358.818,Z 862.503,A -85,B 0,C 180,E1 9739.24,E2 9739.24} C_VEL
LIN {X 0,Y 362.119,Z 839.726,A -85,B 0,C 180,E1 9738.837,E2 9738.837} C_VEL
LIN {X 0,Y 377.951,Z 680.057,A -85,B 0,C 180,E1 9736.444,E2 9736.444} C_VEL
LIN {X 0,Y 375.278,Z 673.164,A -85,B 0,C 180,E1 9734.229,E2 9734.229} C_VEL
LIN {X 0,Y 372.878,Z 667.25,A -85,B 0,C 180,E1 9731.827,E2 9731.827} C_VEL
LIN {X 0,Y 370.93,Z 662.413,A -85,B 0,C 180,E1 9729.308,E2 9729.308} C_VEL
LIN {X 0,Y 369.221,Z 657.879,A -85,B 0,C 180,E1 9725.907,E2 9725.907} C_VEL
LIN {X 0,Y 368.53,Z 655.567,A -85,B 0,C 180,E1 9721.244,E2 9721.244} C_VEL
LIN {X 0,Y 368.998,Z 656.106,A -85,B 0,C 180,E1 9718.603,E2 9718.603} C_VEL
LIN {X 0,Y 370.86,Z 659.355,A -85,B 0,C 180,E1 9714.663,E2 9714.663} C_VEL
LIN {X 0,Y 373.05,Z 663.696,A -85,B 0,C 180,E1 9711.833,E2 9711.833} C_VEL
